// TIA Portal V18 export
// export: Created 2026-06-07T17:38:19.8064699Z, ExportSetting WithDefaults, DisplayName Totally Integrated Automation Portal, DisplayVersion V18, DisplayName TIA Portal Openness, DisplayVersion V18, DisplayName TIA Portal Version Control Interface, DisplayVersion V18, DisplayName STEP 7 Professional, DisplayVersion V18, DisplayName STEP 7 Safety, DisplayVersion V18, DisplayName WinCC Professional, DisplayVersion V18
FUNCTION "FC_PLC2_Mixing" : Void   // FC20, LAD
{ S7_Optimized_Access := 'TRUE' }
VERSION : 0.1
// stored: AutoNumber true, IsIECCheckEnabled false, SetENOAutomatically false, UDAEnableTagReadback false
BEGIN

REGION Network 1: Khóa nút nhấn Start HMI qua Run Enable PLC2
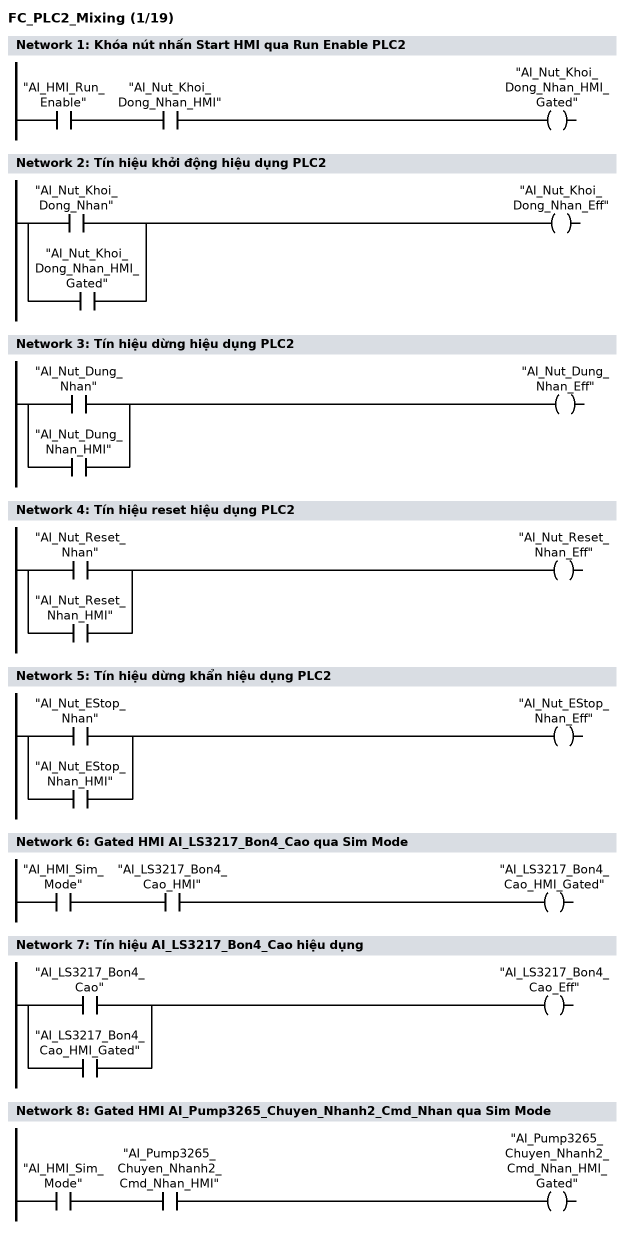
   RUNG wire#powerrail
      Contact( "AI_HMI_Run_Enable" )
      Contact( "AI_Nut_Khoi_Dong_Nhan_HMI" )
      Coil( "AI_Nut_Khoi_Dong_Nhan_HMI_Gated" )
   END_RUNG
   // the same network as SCL:
   "AI_Nut_Khoi_Dong_Nhan_HMI_Gated" := "AI_HMI_Run_Enable" AND "AI_Nut_Khoi_Dong_Nhan_HMI";
END_REGION

REGION Network 2: Tín hiệu khởi động hiệu dụng PLC2
   RUNG wire#powerrail
      Contact( "AI_Nut_Khoi_Dong_Nhan" )
      wire#w1
      Coil( "AI_Nut_Khoi_Dong_Nhan_Eff" )
   END_RUNG
   RUNG wire#powerrail
      Contact( "AI_Nut_Khoi_Dong_Nhan_HMI_Gated" )
   END_RUNG wire#w1
   // the same network as SCL:
   "AI_Nut_Khoi_Dong_Nhan_Eff" := "AI_Nut_Khoi_Dong_Nhan" OR "AI_Nut_Khoi_Dong_Nhan_HMI_Gated";
END_REGION

REGION Network 3: Tín hiệu dừng hiệu dụng PLC2
   RUNG wire#powerrail
      Contact( "AI_Nut_Dung_Nhan" )
      wire#w1
      Coil( "AI_Nut_Dung_Nhan_Eff" )
   END_RUNG
   RUNG wire#powerrail
      Contact( "AI_Nut_Dung_Nhan_HMI" )
   END_RUNG wire#w1
   // the same network as SCL:
   "AI_Nut_Dung_Nhan_Eff" := "AI_Nut_Dung_Nhan" OR "AI_Nut_Dung_Nhan_HMI";
END_REGION

REGION Network 4: Tín hiệu reset hiệu dụng PLC2
   RUNG wire#powerrail
      Contact( "AI_Nut_Reset_Nhan" )
      wire#w1
      Coil( "AI_Nut_Reset_Nhan_Eff" )
   END_RUNG
   RUNG wire#powerrail
      Contact( "AI_Nut_Reset_Nhan_HMI" )
   END_RUNG wire#w1
   // the same network as SCL:
   "AI_Nut_Reset_Nhan_Eff" := "AI_Nut_Reset_Nhan" OR "AI_Nut_Reset_Nhan_HMI";
END_REGION

REGION Network 5: Tín hiệu dừng khẩn hiệu dụng PLC2
   RUNG wire#powerrail
      Contact( "AI_Nut_EStop_Nhan" )
      wire#w1
      Coil( "AI_Nut_EStop_Nhan_Eff" )
   END_RUNG
   RUNG wire#powerrail
      Contact( "AI_Nut_EStop_Nhan_HMI" )
   END_RUNG wire#w1
   // the same network as SCL:
   "AI_Nut_EStop_Nhan_Eff" := "AI_Nut_EStop_Nhan" OR "AI_Nut_EStop_Nhan_HMI";
END_REGION

REGION Network 6: Gated HMI AI_LS3217_Bon4_Cao qua Sim Mode
   RUNG wire#powerrail
      Contact( "AI_HMI_Sim_Mode" )
      Contact( "AI_LS3217_Bon4_Cao_HMI" )
      Coil( "AI_LS3217_Bon4_Cao_HMI_Gated" )
   END_RUNG
   // the same network as SCL:
   "AI_LS3217_Bon4_Cao_HMI_Gated" := "AI_HMI_Sim_Mode" AND "AI_LS3217_Bon4_Cao_HMI";
END_REGION

REGION Network 7: Tín hiệu AI_LS3217_Bon4_Cao hiệu dụng
   RUNG wire#powerrail
      Contact( "AI_LS3217_Bon4_Cao" )
      wire#w1
      Coil( "AI_LS3217_Bon4_Cao_Eff" )
   END_RUNG
   RUNG wire#powerrail
      Contact( "AI_LS3217_Bon4_Cao_HMI_Gated" )
   END_RUNG wire#w1
   // the same network as SCL:
   "AI_LS3217_Bon4_Cao_Eff" := "AI_LS3217_Bon4_Cao" OR "AI_LS3217_Bon4_Cao_HMI_Gated";
END_REGION

REGION Network 8: Gated HMI AI_Pump3265_Chuyen_Nhanh2_Cmd_Nhan qua Sim Mode
   RUNG wire#powerrail
      Contact( "AI_HMI_Sim_Mode" )
      Contact( "AI_Pump3265_Chuyen_Nhanh2_Cmd_Nhan_HMI" )
      Coil( "AI_Pump3265_Chuyen_Nhanh2_Cmd_Nhan_HMI_Gated" )
   END_RUNG
   // the same network as SCL:
   "AI_Pump3265_Chuyen_Nhanh2_Cmd_Nhan_HMI_Gated" := "AI_HMI_Sim_Mode" AND "AI_Pump3265_Chuyen_Nhanh2_Cmd_Nhan_HMI";
END_REGION

REGION Network 9: Tín hiệu AI_Pump3265_Chuyen_Nhanh2_Cmd_Nhan hiệu dụng
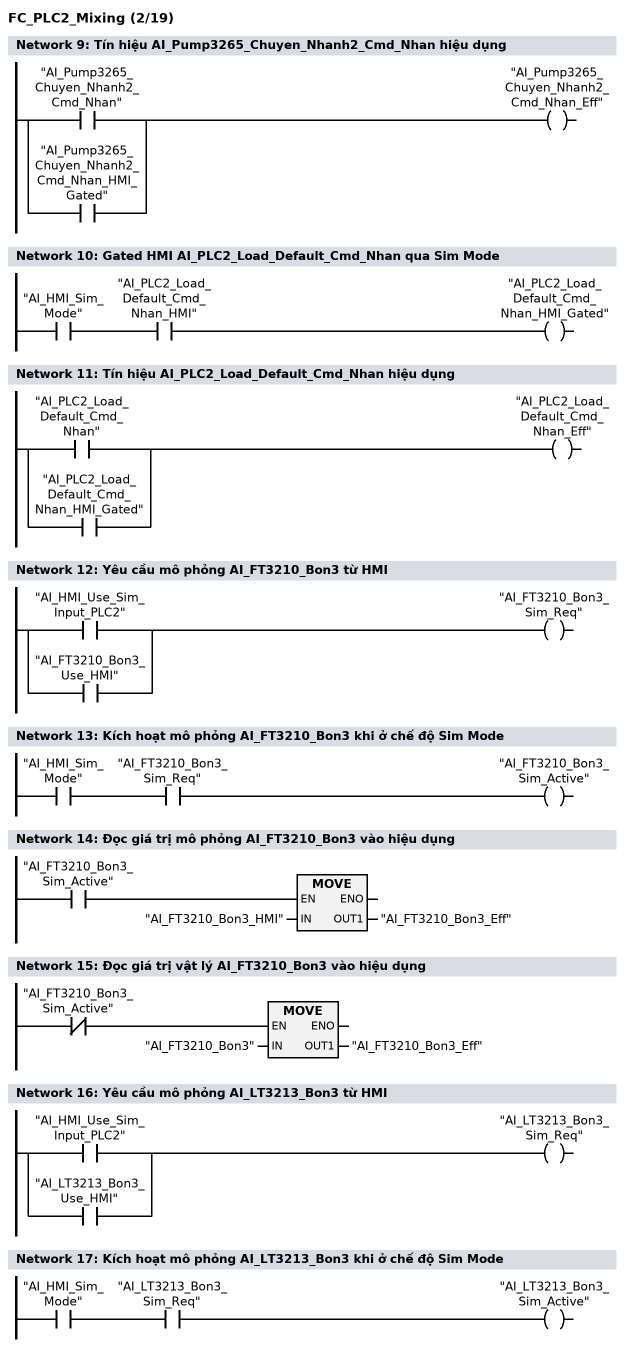
   RUNG wire#powerrail
      Contact( "AI_Pump3265_Chuyen_Nhanh2_Cmd_Nhan" )
      wire#w1
      Coil( "AI_Pump3265_Chuyen_Nhanh2_Cmd_Nhan_Eff" )
   END_RUNG
   RUNG wire#powerrail
      Contact( "AI_Pump3265_Chuyen_Nhanh2_Cmd_Nhan_HMI_Gated" )
   END_RUNG wire#w1
   // the same network as SCL:
   "AI_Pump3265_Chuyen_Nhanh2_Cmd_Nhan_Eff" := "AI_Pump3265_Chuyen_Nhanh2_Cmd_Nhan" OR "AI_Pump3265_Chuyen_Nhanh2_Cmd_Nhan_HMI_Gated";
END_REGION

REGION Network 10: Gated HMI AI_PLC2_Load_Default_Cmd_Nhan qua Sim Mode
   RUNG wire#powerrail
      Contact( "AI_HMI_Sim_Mode" )
      Contact( "AI_PLC2_Load_Default_Cmd_Nhan_HMI" )
      Coil( "AI_PLC2_Load_Default_Cmd_Nhan_HMI_Gated" )
   END_RUNG
   // the same network as SCL:
   "AI_PLC2_Load_Default_Cmd_Nhan_HMI_Gated" := "AI_HMI_Sim_Mode" AND "AI_PLC2_Load_Default_Cmd_Nhan_HMI";
END_REGION

REGION Network 11: Tín hiệu AI_PLC2_Load_Default_Cmd_Nhan hiệu dụng
   RUNG wire#powerrail
      Contact( "AI_PLC2_Load_Default_Cmd_Nhan" )
      wire#w1
      Coil( "AI_PLC2_Load_Default_Cmd_Nhan_Eff" )
   END_RUNG
   RUNG wire#powerrail
      Contact( "AI_PLC2_Load_Default_Cmd_Nhan_HMI_Gated" )
   END_RUNG wire#w1
   // the same network as SCL:
   "AI_PLC2_Load_Default_Cmd_Nhan_Eff" := "AI_PLC2_Load_Default_Cmd_Nhan" OR "AI_PLC2_Load_Default_Cmd_Nhan_HMI_Gated";
END_REGION

REGION Network 12: Yêu cầu mô phỏng AI_FT3210_Bon3 từ HMI
   RUNG wire#powerrail
      Contact( "AI_HMI_Use_Sim_Input_PLC2" )
      wire#w1
      Coil( "AI_FT3210_Bon3_Sim_Req" )
   END_RUNG
   RUNG wire#powerrail
      Contact( "AI_FT3210_Bon3_Use_HMI" )
   END_RUNG wire#w1
   // the same network as SCL:
   "AI_FT3210_Bon3_Sim_Req" := "AI_HMI_Use_Sim_Input_PLC2" OR "AI_FT3210_Bon3_Use_HMI";
END_REGION

REGION Network 13: Kích hoạt mô phỏng AI_FT3210_Bon3 khi ở chế độ Sim Mode
   RUNG wire#powerrail
      Contact( "AI_HMI_Sim_Mode" )
      Contact( "AI_FT3210_Bon3_Sim_Req" )
      Coil( "AI_FT3210_Bon3_Sim_Active" )
   END_RUNG
   // the same network as SCL:
   "AI_FT3210_Bon3_Sim_Active" := "AI_HMI_Sim_Mode" AND "AI_FT3210_Bon3_Sim_Req";
END_REGION

REGION Network 14: Đọc giá trị mô phỏng AI_FT3210_Bon3 vào hiệu dụng
   RUNG wire#powerrail
      Contact( "AI_FT3210_Bon3_Sim_Active" )
      { S7_GenerateENO := "TRUE" } Move(in := "AI_FT3210_Bon3_HMI", out1 => "AI_FT3210_Bon3_Eff")
   END_RUNG
   // the same network as SCL:
   IF "AI_FT3210_Bon3_Sim_Active" THEN "AI_FT3210_Bon3_Eff" := "AI_FT3210_Bon3_HMI"; END_IF;
END_REGION

REGION Network 15: Đọc giá trị vật lý AI_FT3210_Bon3 vào hiệu dụng
   RUNG wire#powerrail
      I_Contact( "AI_FT3210_Bon3_Sim_Active" )
      { S7_GenerateENO := "TRUE" } Move(in := "AI_FT3210_Bon3", out1 => "AI_FT3210_Bon3_Eff")
   END_RUNG
   // the same network as SCL:
   IF NOT "AI_FT3210_Bon3_Sim_Active" THEN "AI_FT3210_Bon3_Eff" := "AI_FT3210_Bon3"; END_IF;
END_REGION

REGION Network 16: Yêu cầu mô phỏng AI_LT3213_Bon3 từ HMI
   RUNG wire#powerrail
      Contact( "AI_HMI_Use_Sim_Input_PLC2" )
      wire#w1
      Coil( "AI_LT3213_Bon3_Sim_Req" )
   END_RUNG
   RUNG wire#powerrail
      Contact( "AI_LT3213_Bon3_Use_HMI" )
   END_RUNG wire#w1
   // the same network as SCL:
   "AI_LT3213_Bon3_Sim_Req" := "AI_HMI_Use_Sim_Input_PLC2" OR "AI_LT3213_Bon3_Use_HMI";
END_REGION

REGION Network 17: Kích hoạt mô phỏng AI_LT3213_Bon3 khi ở chế độ Sim Mode
   RUNG wire#powerrail
      Contact( "AI_HMI_Sim_Mode" )
      Contact( "AI_LT3213_Bon3_Sim_Req" )
      Coil( "AI_LT3213_Bon3_Sim_Active" )
   END_RUNG
   // the same network as SCL:
   "AI_LT3213_Bon3_Sim_Active" := "AI_HMI_Sim_Mode" AND "AI_LT3213_Bon3_Sim_Req";
END_REGION

REGION Network 18: Đọc giá trị mô phỏng AI_LT3213_Bon3 vào hiệu dụng
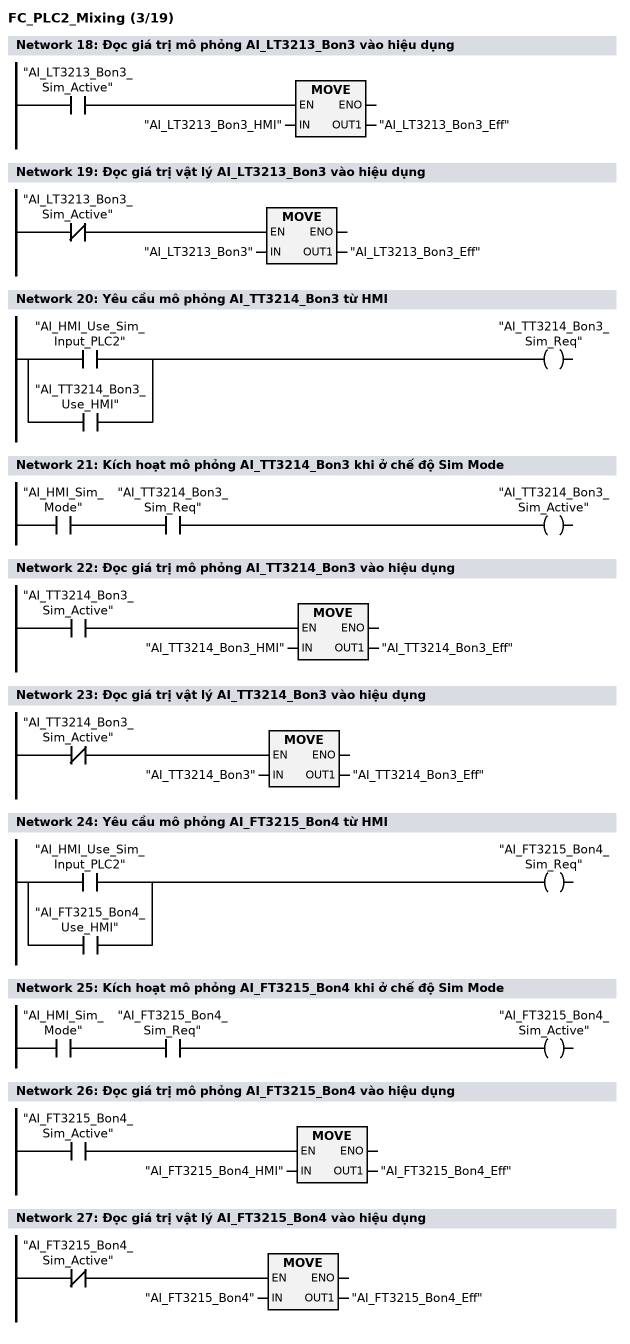
   RUNG wire#powerrail
      Contact( "AI_LT3213_Bon3_Sim_Active" )
      { S7_GenerateENO := "TRUE" } Move(in := "AI_LT3213_Bon3_HMI", out1 => "AI_LT3213_Bon3_Eff")
   END_RUNG
   // the same network as SCL:
   IF "AI_LT3213_Bon3_Sim_Active" THEN "AI_LT3213_Bon3_Eff" := "AI_LT3213_Bon3_HMI"; END_IF;
END_REGION

REGION Network 19: Đọc giá trị vật lý AI_LT3213_Bon3 vào hiệu dụng
   RUNG wire#powerrail
      I_Contact( "AI_LT3213_Bon3_Sim_Active" )
      { S7_GenerateENO := "TRUE" } Move(in := "AI_LT3213_Bon3", out1 => "AI_LT3213_Bon3_Eff")
   END_RUNG
   // the same network as SCL:
   IF NOT "AI_LT3213_Bon3_Sim_Active" THEN "AI_LT3213_Bon3_Eff" := "AI_LT3213_Bon3"; END_IF;
END_REGION

REGION Network 20: Yêu cầu mô phỏng AI_TT3214_Bon3 từ HMI
   RUNG wire#powerrail
      Contact( "AI_HMI_Use_Sim_Input_PLC2" )
      wire#w1
      Coil( "AI_TT3214_Bon3_Sim_Req" )
   END_RUNG
   RUNG wire#powerrail
      Contact( "AI_TT3214_Bon3_Use_HMI" )
   END_RUNG wire#w1
   // the same network as SCL:
   "AI_TT3214_Bon3_Sim_Req" := "AI_HMI_Use_Sim_Input_PLC2" OR "AI_TT3214_Bon3_Use_HMI";
END_REGION

REGION Network 21: Kích hoạt mô phỏng AI_TT3214_Bon3 khi ở chế độ Sim Mode
   RUNG wire#powerrail
      Contact( "AI_HMI_Sim_Mode" )
      Contact( "AI_TT3214_Bon3_Sim_Req" )
      Coil( "AI_TT3214_Bon3_Sim_Active" )
   END_RUNG
   // the same network as SCL:
   "AI_TT3214_Bon3_Sim_Active" := "AI_HMI_Sim_Mode" AND "AI_TT3214_Bon3_Sim_Req";
END_REGION

REGION Network 22: Đọc giá trị mô phỏng AI_TT3214_Bon3 vào hiệu dụng
   RUNG wire#powerrail
      Contact( "AI_TT3214_Bon3_Sim_Active" )
      { S7_GenerateENO := "TRUE" } Move(in := "AI_TT3214_Bon3_HMI", out1 => "AI_TT3214_Bon3_Eff")
   END_RUNG
   // the same network as SCL:
   IF "AI_TT3214_Bon3_Sim_Active" THEN "AI_TT3214_Bon3_Eff" := "AI_TT3214_Bon3_HMI"; END_IF;
END_REGION

REGION Network 23: Đọc giá trị vật lý AI_TT3214_Bon3 vào hiệu dụng
   RUNG wire#powerrail
      I_Contact( "AI_TT3214_Bon3_Sim_Active" )
      { S7_GenerateENO := "TRUE" } Move(in := "AI_TT3214_Bon3", out1 => "AI_TT3214_Bon3_Eff")
   END_RUNG
   // the same network as SCL:
   IF NOT "AI_TT3214_Bon3_Sim_Active" THEN "AI_TT3214_Bon3_Eff" := "AI_TT3214_Bon3"; END_IF;
END_REGION

REGION Network 24: Yêu cầu mô phỏng AI_FT3215_Bon4 từ HMI
   RUNG wire#powerrail
      Contact( "AI_HMI_Use_Sim_Input_PLC2" )
      wire#w1
      Coil( "AI_FT3215_Bon4_Sim_Req" )
   END_RUNG
   RUNG wire#powerrail
      Contact( "AI_FT3215_Bon4_Use_HMI" )
   END_RUNG wire#w1
   // the same network as SCL:
   "AI_FT3215_Bon4_Sim_Req" := "AI_HMI_Use_Sim_Input_PLC2" OR "AI_FT3215_Bon4_Use_HMI";
END_REGION

REGION Network 25: Kích hoạt mô phỏng AI_FT3215_Bon4 khi ở chế độ Sim Mode
   RUNG wire#powerrail
      Contact( "AI_HMI_Sim_Mode" )
      Contact( "AI_FT3215_Bon4_Sim_Req" )
      Coil( "AI_FT3215_Bon4_Sim_Active" )
   END_RUNG
   // the same network as SCL:
   "AI_FT3215_Bon4_Sim_Active" := "AI_HMI_Sim_Mode" AND "AI_FT3215_Bon4_Sim_Req";
END_REGION

REGION Network 26: Đọc giá trị mô phỏng AI_FT3215_Bon4 vào hiệu dụng
   RUNG wire#powerrail
      Contact( "AI_FT3215_Bon4_Sim_Active" )
      { S7_GenerateENO := "TRUE" } Move(in := "AI_FT3215_Bon4_HMI", out1 => "AI_FT3215_Bon4_Eff")
   END_RUNG
   // the same network as SCL:
   IF "AI_FT3215_Bon4_Sim_Active" THEN "AI_FT3215_Bon4_Eff" := "AI_FT3215_Bon4_HMI"; END_IF;
END_REGION

REGION Network 27: Đọc giá trị vật lý AI_FT3215_Bon4 vào hiệu dụng
   RUNG wire#powerrail
      I_Contact( "AI_FT3215_Bon4_Sim_Active" )
      { S7_GenerateENO := "TRUE" } Move(in := "AI_FT3215_Bon4", out1 => "AI_FT3215_Bon4_Eff")
   END_RUNG
   // the same network as SCL:
   IF NOT "AI_FT3215_Bon4_Sim_Active" THEN "AI_FT3215_Bon4_Eff" := "AI_FT3215_Bon4"; END_IF;
END_REGION

REGION Network 28: Yêu cầu mô phỏng AI_FQ3215_Bon4 từ HMI
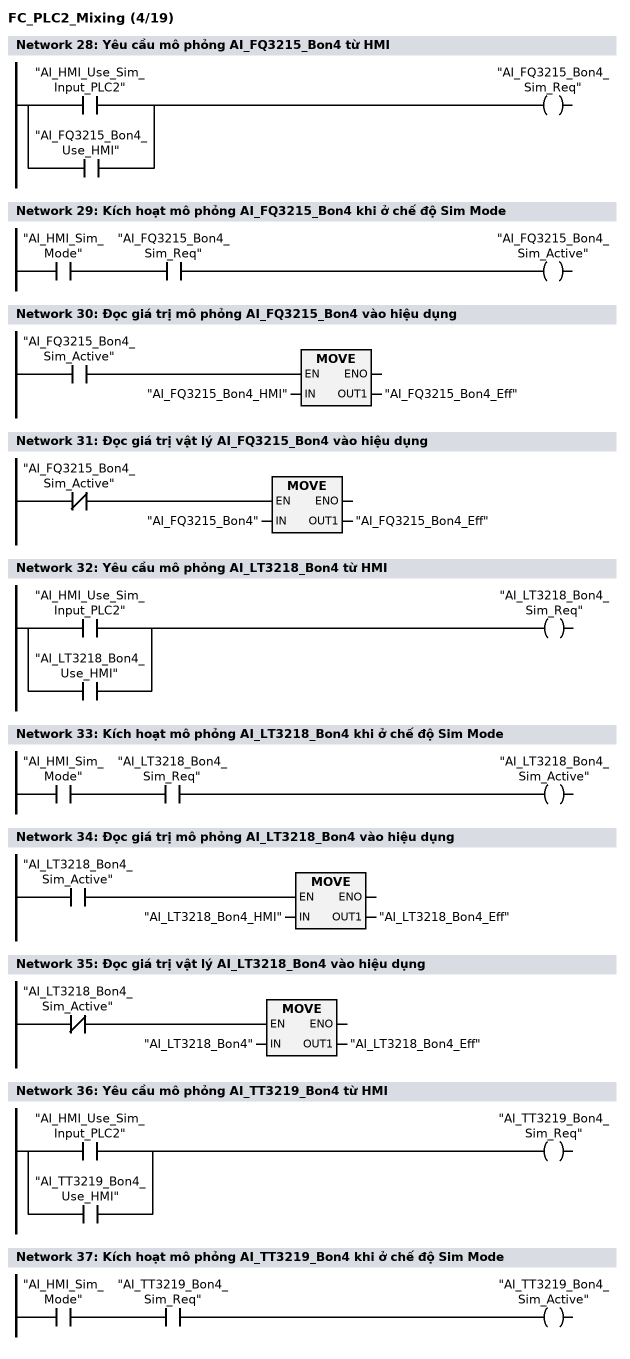
   RUNG wire#powerrail
      Contact( "AI_HMI_Use_Sim_Input_PLC2" )
      wire#w1
      Coil( "AI_FQ3215_Bon4_Sim_Req" )
   END_RUNG
   RUNG wire#powerrail
      Contact( "AI_FQ3215_Bon4_Use_HMI" )
   END_RUNG wire#w1
   // the same network as SCL:
   "AI_FQ3215_Bon4_Sim_Req" := "AI_HMI_Use_Sim_Input_PLC2" OR "AI_FQ3215_Bon4_Use_HMI";
END_REGION

REGION Network 29: Kích hoạt mô phỏng AI_FQ3215_Bon4 khi ở chế độ Sim Mode
   RUNG wire#powerrail
      Contact( "AI_HMI_Sim_Mode" )
      Contact( "AI_FQ3215_Bon4_Sim_Req" )
      Coil( "AI_FQ3215_Bon4_Sim_Active" )
   END_RUNG
   // the same network as SCL:
   "AI_FQ3215_Bon4_Sim_Active" := "AI_HMI_Sim_Mode" AND "AI_FQ3215_Bon4_Sim_Req";
END_REGION

REGION Network 30: Đọc giá trị mô phỏng AI_FQ3215_Bon4 vào hiệu dụng
   RUNG wire#powerrail
      Contact( "AI_FQ3215_Bon4_Sim_Active" )
      { S7_GenerateENO := "TRUE" } Move(in := "AI_FQ3215_Bon4_HMI", out1 => "AI_FQ3215_Bon4_Eff")
   END_RUNG
   // the same network as SCL:
   IF "AI_FQ3215_Bon4_Sim_Active" THEN "AI_FQ3215_Bon4_Eff" := "AI_FQ3215_Bon4_HMI"; END_IF;
END_REGION

REGION Network 31: Đọc giá trị vật lý AI_FQ3215_Bon4 vào hiệu dụng
   RUNG wire#powerrail
      I_Contact( "AI_FQ3215_Bon4_Sim_Active" )
      { S7_GenerateENO := "TRUE" } Move(in := "AI_FQ3215_Bon4", out1 => "AI_FQ3215_Bon4_Eff")
   END_RUNG
   // the same network as SCL:
   IF NOT "AI_FQ3215_Bon4_Sim_Active" THEN "AI_FQ3215_Bon4_Eff" := "AI_FQ3215_Bon4"; END_IF;
END_REGION

REGION Network 32: Yêu cầu mô phỏng AI_LT3218_Bon4 từ HMI
   RUNG wire#powerrail
      Contact( "AI_HMI_Use_Sim_Input_PLC2" )
      wire#w1
      Coil( "AI_LT3218_Bon4_Sim_Req" )
   END_RUNG
   RUNG wire#powerrail
      Contact( "AI_LT3218_Bon4_Use_HMI" )
   END_RUNG wire#w1
   // the same network as SCL:
   "AI_LT3218_Bon4_Sim_Req" := "AI_HMI_Use_Sim_Input_PLC2" OR "AI_LT3218_Bon4_Use_HMI";
END_REGION

REGION Network 33: Kích hoạt mô phỏng AI_LT3218_Bon4 khi ở chế độ Sim Mode
   RUNG wire#powerrail
      Contact( "AI_HMI_Sim_Mode" )
      Contact( "AI_LT3218_Bon4_Sim_Req" )
      Coil( "AI_LT3218_Bon4_Sim_Active" )
   END_RUNG
   // the same network as SCL:
   "AI_LT3218_Bon4_Sim_Active" := "AI_HMI_Sim_Mode" AND "AI_LT3218_Bon4_Sim_Req";
END_REGION

REGION Network 34: Đọc giá trị mô phỏng AI_LT3218_Bon4 vào hiệu dụng
   RUNG wire#powerrail
      Contact( "AI_LT3218_Bon4_Sim_Active" )
      { S7_GenerateENO := "TRUE" } Move(in := "AI_LT3218_Bon4_HMI", out1 => "AI_LT3218_Bon4_Eff")
   END_RUNG
   // the same network as SCL:
   IF "AI_LT3218_Bon4_Sim_Active" THEN "AI_LT3218_Bon4_Eff" := "AI_LT3218_Bon4_HMI"; END_IF;
END_REGION

REGION Network 35: Đọc giá trị vật lý AI_LT3218_Bon4 vào hiệu dụng
   RUNG wire#powerrail
      I_Contact( "AI_LT3218_Bon4_Sim_Active" )
      { S7_GenerateENO := "TRUE" } Move(in := "AI_LT3218_Bon4", out1 => "AI_LT3218_Bon4_Eff")
   END_RUNG
   // the same network as SCL:
   IF NOT "AI_LT3218_Bon4_Sim_Active" THEN "AI_LT3218_Bon4_Eff" := "AI_LT3218_Bon4"; END_IF;
END_REGION

REGION Network 36: Yêu cầu mô phỏng AI_TT3219_Bon4 từ HMI
   RUNG wire#powerrail
      Contact( "AI_HMI_Use_Sim_Input_PLC2" )
      wire#w1
      Coil( "AI_TT3219_Bon4_Sim_Req" )
   END_RUNG
   RUNG wire#powerrail
      Contact( "AI_TT3219_Bon4_Use_HMI" )
   END_RUNG wire#w1
   // the same network as SCL:
   "AI_TT3219_Bon4_Sim_Req" := "AI_HMI_Use_Sim_Input_PLC2" OR "AI_TT3219_Bon4_Use_HMI";
END_REGION

REGION Network 37: Kích hoạt mô phỏng AI_TT3219_Bon4 khi ở chế độ Sim Mode
   RUNG wire#powerrail
      Contact( "AI_HMI_Sim_Mode" )
      Contact( "AI_TT3219_Bon4_Sim_Req" )
      Coil( "AI_TT3219_Bon4_Sim_Active" )
   END_RUNG
   // the same network as SCL:
   "AI_TT3219_Bon4_Sim_Active" := "AI_HMI_Sim_Mode" AND "AI_TT3219_Bon4_Sim_Req";
END_REGION

REGION Network 38: Đọc giá trị mô phỏng AI_TT3219_Bon4 vào hiệu dụng
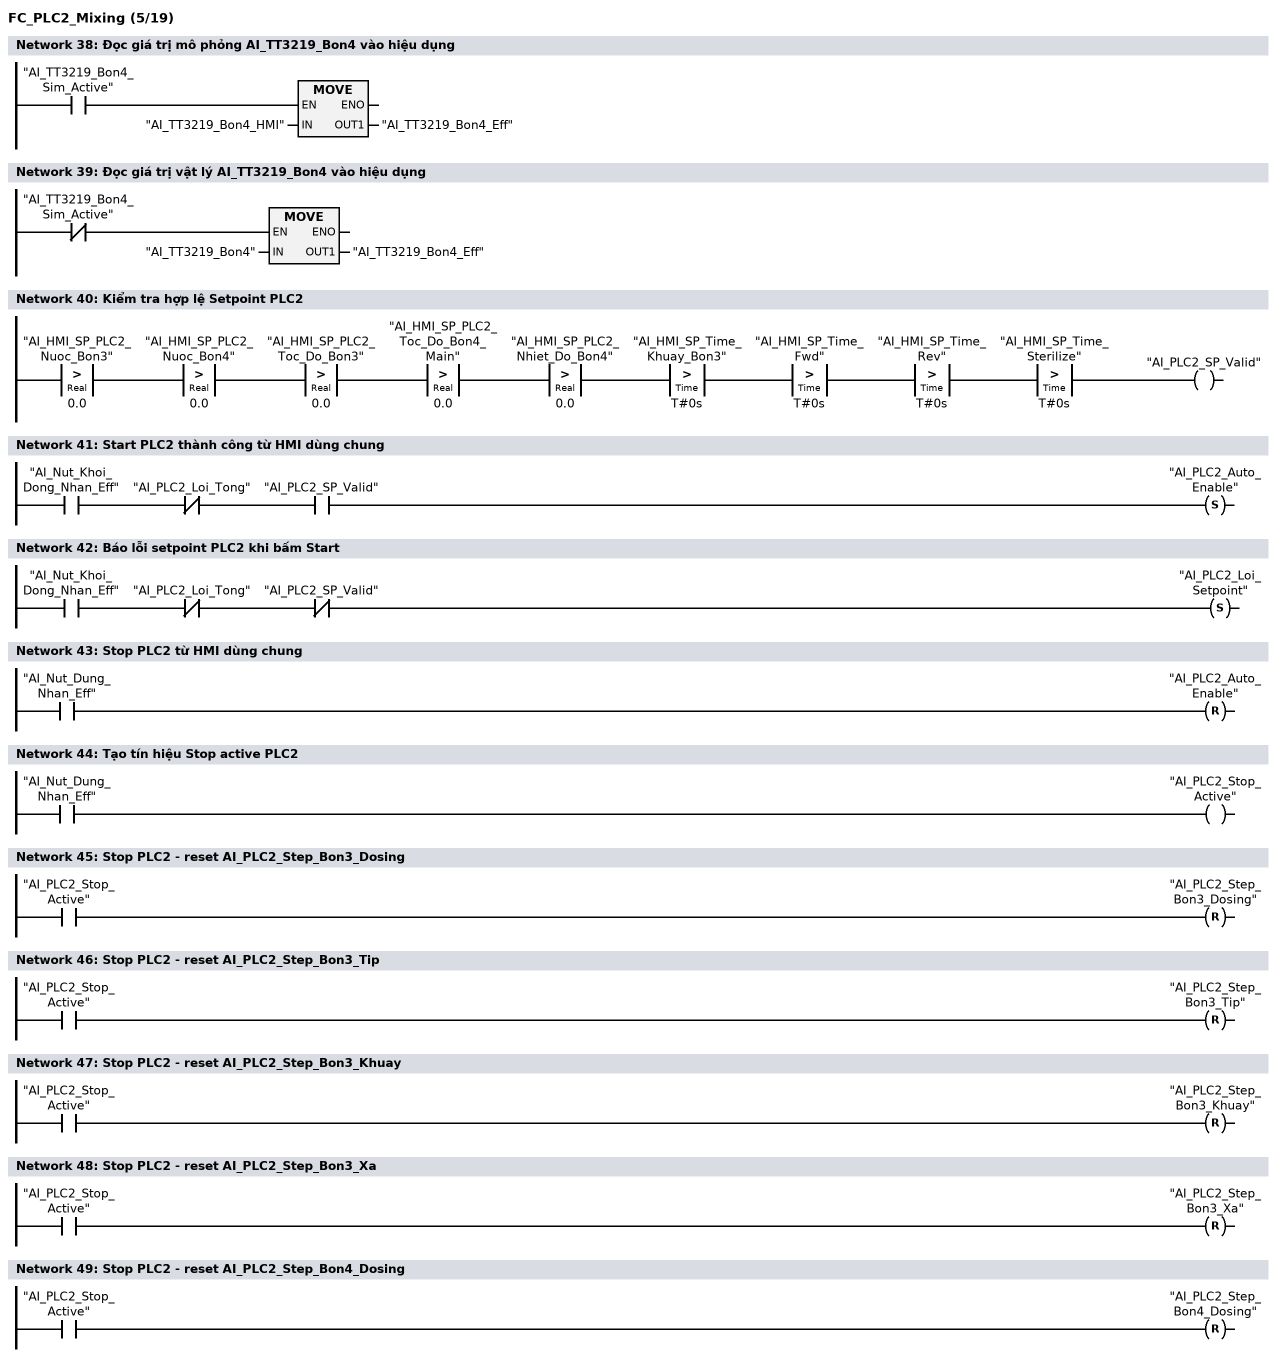
   RUNG wire#powerrail
      Contact( "AI_TT3219_Bon4_Sim_Active" )
      { S7_GenerateENO := "TRUE" } Move(in := "AI_TT3219_Bon4_HMI", out1 => "AI_TT3219_Bon4_Eff")
   END_RUNG
   // the same network as SCL:
   IF "AI_TT3219_Bon4_Sim_Active" THEN "AI_TT3219_Bon4_Eff" := "AI_TT3219_Bon4_HMI"; END_IF;
END_REGION

REGION Network 39: Đọc giá trị vật lý AI_TT3219_Bon4 vào hiệu dụng
   RUNG wire#powerrail
      I_Contact( "AI_TT3219_Bon4_Sim_Active" )
      { S7_GenerateENO := "TRUE" } Move(in := "AI_TT3219_Bon4", out1 => "AI_TT3219_Bon4_Eff")
   END_RUNG
   // the same network as SCL:
   IF NOT "AI_TT3219_Bon4_Sim_Active" THEN "AI_TT3219_Bon4_Eff" := "AI_TT3219_Bon4"; END_IF;
END_REGION

REGION Network 40: Kiểm tra hợp lệ Setpoint PLC2
   RUNG wire#powerrail
      { S7_Templates := "SrcType := Real" } GT_Contact(in1 := "AI_HMI_SP_PLC2_Nuoc_Bon3", in2 := 0.0)
      { S7_Templates := "SrcType := Real" } GT_Contact(in1 := "AI_HMI_SP_PLC2_Nuoc_Bon4", in2 := 0.0)
      { S7_Templates := "SrcType := Real" } GT_Contact(in1 := "AI_HMI_SP_PLC2_Toc_Do_Bon3", in2 := 0.0)
      { S7_Templates := "SrcType := Real" } GT_Contact(in1 := "AI_HMI_SP_PLC2_Toc_Do_Bon4_Main", in2 := 0.0)
      { S7_Templates := "SrcType := Real" } GT_Contact(in1 := "AI_HMI_SP_PLC2_Nhiet_Do_Bon4", in2 := 0.0)
      { S7_Templates := "SrcType := Time" } GT_Contact(in1 := "AI_HMI_SP_Time_Khuay_Bon3", in2 := T#0s)
      { S7_Templates := "SrcType := Time" } GT_Contact(in1 := "AI_HMI_SP_Time_Fwd", in2 := T#0s)
      { S7_Templates := "SrcType := Time" } GT_Contact(in1 := "AI_HMI_SP_Time_Rev", in2 := T#0s)
      { S7_Templates := "SrcType := Time" } GT_Contact(in1 := "AI_HMI_SP_Time_Sterilize", in2 := T#0s)
      Coil( "AI_PLC2_SP_Valid" )
   END_RUNG
   // the same network as SCL:
   "AI_PLC2_SP_Valid" := ("AI_HMI_SP_PLC2_Nuoc_Bon3" > 0.0) AND ("AI_HMI_SP_PLC2_Nuoc_Bon4" > 0.0) AND ("AI_HMI_SP_PLC2_Toc_Do_Bon3" > 0.0) AND ("AI_HMI_SP_PLC2_Toc_Do_Bon4_Main" > 0.0) AND ("AI_HMI_SP_PLC2_Nhiet_Do_Bon4" > 0.0) AND ("AI_HMI_SP_Time_Khuay_Bon3" > T#0s) AND ("AI_HMI_SP_Time_Fwd" > T#0s) AND ("AI_HMI_SP_Time_Rev" > T#0s) AND ("AI_HMI_SP_Time_Sterilize" > T#0s);
END_REGION

REGION Network 41: Start PLC2 thành công từ HMI dùng chung
   RUNG wire#powerrail
      Contact( "AI_Nut_Khoi_Dong_Nhan_Eff" )
      I_Contact( "AI_PLC2_Loi_Tong" )
      Contact( "AI_PLC2_SP_Valid" )
      S_Coil( "AI_PLC2_Auto_Enable" )
   END_RUNG
   // the same network as SCL:
   IF "AI_Nut_Khoi_Dong_Nhan_Eff" AND NOT "AI_PLC2_Loi_Tong" AND "AI_PLC2_SP_Valid" THEN
       "AI_PLC2_Auto_Enable" := TRUE;
   END_IF;
END_REGION

REGION Network 42: Báo lỗi setpoint PLC2 khi bấm Start
   RUNG wire#powerrail
      Contact( "AI_Nut_Khoi_Dong_Nhan_Eff" )
      I_Contact( "AI_PLC2_Loi_Tong" )
      I_Contact( "AI_PLC2_SP_Valid" )
      S_Coil( "AI_PLC2_Loi_Setpoint" )
   END_RUNG
   // the same network as SCL:
   IF "AI_Nut_Khoi_Dong_Nhan_Eff" AND NOT "AI_PLC2_Loi_Tong" AND NOT "AI_PLC2_SP_Valid" THEN
       "AI_PLC2_Loi_Setpoint" := TRUE;
   END_IF;
END_REGION

REGION Network 43: Stop PLC2 từ HMI dùng chung
   RUNG wire#powerrail
      Contact( "AI_Nut_Dung_Nhan_Eff" )
      R_Coil( "AI_PLC2_Auto_Enable" )
   END_RUNG
   // the same network as SCL:
   IF "AI_Nut_Dung_Nhan_Eff" THEN "AI_PLC2_Auto_Enable" := FALSE; END_IF;
END_REGION

REGION Network 44: Tạo tín hiệu Stop active PLC2
   RUNG wire#powerrail
      Contact( "AI_Nut_Dung_Nhan_Eff" )
      Coil( "AI_PLC2_Stop_Active" )
   END_RUNG
   // the same network as SCL:
   "AI_PLC2_Stop_Active" := "AI_Nut_Dung_Nhan_Eff";
END_REGION

REGION Network 45: Stop PLC2 - reset AI_PLC2_Step_Bon3_Dosing
   RUNG wire#powerrail
      Contact( "AI_PLC2_Stop_Active" )
      R_Coil( "AI_PLC2_Step_Bon3_Dosing" )
   END_RUNG
   // the same network as SCL:
   IF "AI_PLC2_Stop_Active" THEN "AI_PLC2_Step_Bon3_Dosing" := FALSE; END_IF;
END_REGION

REGION Network 46: Stop PLC2 - reset AI_PLC2_Step_Bon3_Tip
   RUNG wire#powerrail
      Contact( "AI_PLC2_Stop_Active" )
      R_Coil( "AI_PLC2_Step_Bon3_Tip" )
   END_RUNG
   // the same network as SCL:
   IF "AI_PLC2_Stop_Active" THEN "AI_PLC2_Step_Bon3_Tip" := FALSE; END_IF;
END_REGION

REGION Network 47: Stop PLC2 - reset AI_PLC2_Step_Bon3_Khuay
   RUNG wire#powerrail
      Contact( "AI_PLC2_Stop_Active" )
      R_Coil( "AI_PLC2_Step_Bon3_Khuay" )
   END_RUNG
   // the same network as SCL:
   IF "AI_PLC2_Stop_Active" THEN "AI_PLC2_Step_Bon3_Khuay" := FALSE; END_IF;
END_REGION

REGION Network 48: Stop PLC2 - reset AI_PLC2_Step_Bon3_Xa
   RUNG wire#powerrail
      Contact( "AI_PLC2_Stop_Active" )
      R_Coil( "AI_PLC2_Step_Bon3_Xa" )
   END_RUNG
   // the same network as SCL:
   IF "AI_PLC2_Stop_Active" THEN "AI_PLC2_Step_Bon3_Xa" := FALSE; END_IF;
END_REGION

REGION Network 49: Stop PLC2 - reset AI_PLC2_Step_Bon4_Dosing
   RUNG wire#powerrail
      Contact( "AI_PLC2_Stop_Active" )
      R_Coil( "AI_PLC2_Step_Bon4_Dosing" )
   END_RUNG
   // the same network as SCL:
   IF "AI_PLC2_Stop_Active" THEN "AI_PLC2_Step_Bon4_Dosing" := FALSE; END_IF;
END_REGION

REGION Network 50: Stop PLC2 - reset AI_PLC2_Step_Bon4_Tip
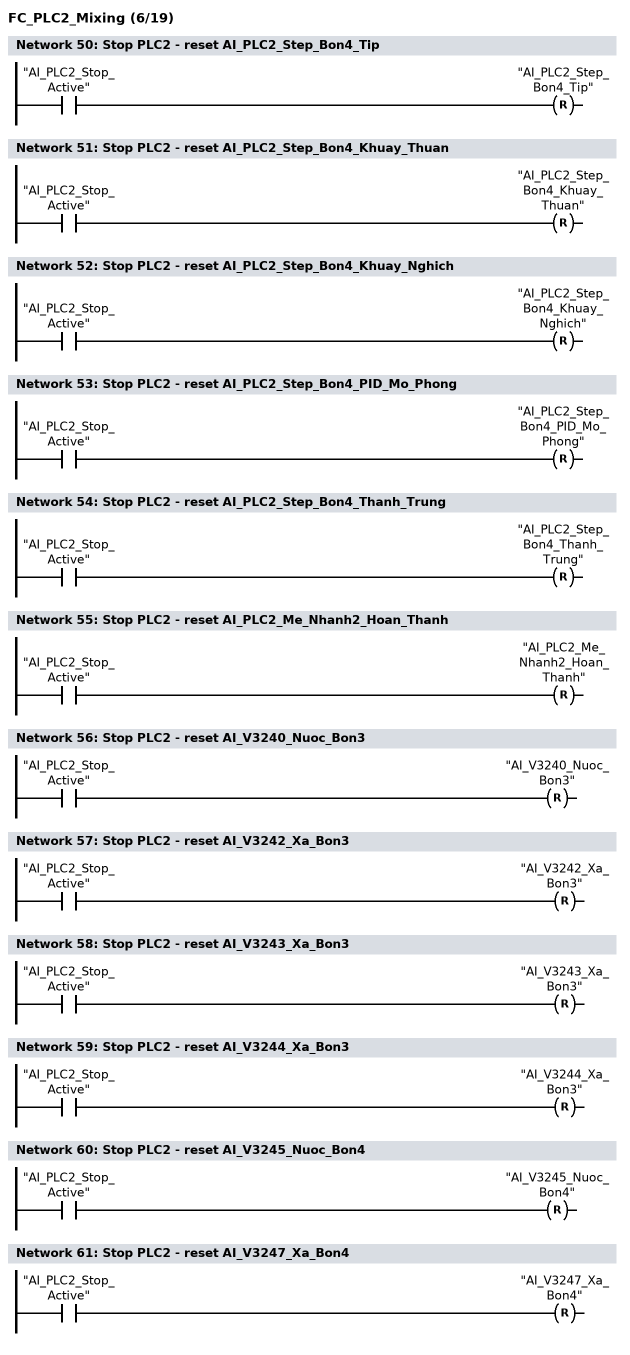
   RUNG wire#powerrail
      Contact( "AI_PLC2_Stop_Active" )
      R_Coil( "AI_PLC2_Step_Bon4_Tip" )
   END_RUNG
   // the same network as SCL:
   IF "AI_PLC2_Stop_Active" THEN "AI_PLC2_Step_Bon4_Tip" := FALSE; END_IF;
END_REGION

REGION Network 51: Stop PLC2 - reset AI_PLC2_Step_Bon4_Khuay_Thuan
   RUNG wire#powerrail
      Contact( "AI_PLC2_Stop_Active" )
      R_Coil( "AI_PLC2_Step_Bon4_Khuay_Thuan" )
   END_RUNG
   // the same network as SCL:
   IF "AI_PLC2_Stop_Active" THEN "AI_PLC2_Step_Bon4_Khuay_Thuan" := FALSE; END_IF;
END_REGION

REGION Network 52: Stop PLC2 - reset AI_PLC2_Step_Bon4_Khuay_Nghich
   RUNG wire#powerrail
      Contact( "AI_PLC2_Stop_Active" )
      R_Coil( "AI_PLC2_Step_Bon4_Khuay_Nghich" )
   END_RUNG
   // the same network as SCL:
   IF "AI_PLC2_Stop_Active" THEN "AI_PLC2_Step_Bon4_Khuay_Nghich" := FALSE; END_IF;
END_REGION

REGION Network 53: Stop PLC2 - reset AI_PLC2_Step_Bon4_PID_Mo_Phong
   RUNG wire#powerrail
      Contact( "AI_PLC2_Stop_Active" )
      R_Coil( "AI_PLC2_Step_Bon4_PID_Mo_Phong" )
   END_RUNG
   // the same network as SCL:
   IF "AI_PLC2_Stop_Active" THEN "AI_PLC2_Step_Bon4_PID_Mo_Phong" := FALSE; END_IF;
END_REGION

REGION Network 54: Stop PLC2 - reset AI_PLC2_Step_Bon4_Thanh_Trung
   RUNG wire#powerrail
      Contact( "AI_PLC2_Stop_Active" )
      R_Coil( "AI_PLC2_Step_Bon4_Thanh_Trung" )
   END_RUNG
   // the same network as SCL:
   IF "AI_PLC2_Stop_Active" THEN "AI_PLC2_Step_Bon4_Thanh_Trung" := FALSE; END_IF;
END_REGION

REGION Network 55: Stop PLC2 - reset AI_PLC2_Me_Nhanh2_Hoan_Thanh
   RUNG wire#powerrail
      Contact( "AI_PLC2_Stop_Active" )
      R_Coil( "AI_PLC2_Me_Nhanh2_Hoan_Thanh" )
   END_RUNG
   // the same network as SCL:
   IF "AI_PLC2_Stop_Active" THEN "AI_PLC2_Me_Nhanh2_Hoan_Thanh" := FALSE; END_IF;
END_REGION

REGION Network 56: Stop PLC2 - reset AI_V3240_Nuoc_Bon3
   RUNG wire#powerrail
      Contact( "AI_PLC2_Stop_Active" )
      R_Coil( "AI_V3240_Nuoc_Bon3" )
   END_RUNG
   // the same network as SCL:
   IF "AI_PLC2_Stop_Active" THEN "AI_V3240_Nuoc_Bon3" := FALSE; END_IF;
END_REGION

REGION Network 57: Stop PLC2 - reset AI_V3242_Xa_Bon3
   RUNG wire#powerrail
      Contact( "AI_PLC2_Stop_Active" )
      R_Coil( "AI_V3242_Xa_Bon3" )
   END_RUNG
   // the same network as SCL:
   IF "AI_PLC2_Stop_Active" THEN "AI_V3242_Xa_Bon3" := FALSE; END_IF;
END_REGION

REGION Network 58: Stop PLC2 - reset AI_V3243_Xa_Bon3
   RUNG wire#powerrail
      Contact( "AI_PLC2_Stop_Active" )
      R_Coil( "AI_V3243_Xa_Bon3" )
   END_RUNG
   // the same network as SCL:
   IF "AI_PLC2_Stop_Active" THEN "AI_V3243_Xa_Bon3" := FALSE; END_IF;
END_REGION

REGION Network 59: Stop PLC2 - reset AI_V3244_Xa_Bon3
   RUNG wire#powerrail
      Contact( "AI_PLC2_Stop_Active" )
      R_Coil( "AI_V3244_Xa_Bon3" )
   END_RUNG
   // the same network as SCL:
   IF "AI_PLC2_Stop_Active" THEN "AI_V3244_Xa_Bon3" := FALSE; END_IF;
END_REGION

REGION Network 60: Stop PLC2 - reset AI_V3245_Nuoc_Bon4
   RUNG wire#powerrail
      Contact( "AI_PLC2_Stop_Active" )
      R_Coil( "AI_V3245_Nuoc_Bon4" )
   END_RUNG
   // the same network as SCL:
   IF "AI_PLC2_Stop_Active" THEN "AI_V3245_Nuoc_Bon4" := FALSE; END_IF;
END_REGION

REGION Network 61: Stop PLC2 - reset AI_V3247_Xa_Bon4
   RUNG wire#powerrail
      Contact( "AI_PLC2_Stop_Active" )
      R_Coil( "AI_V3247_Xa_Bon4" )
   END_RUNG
   // the same network as SCL:
   IF "AI_PLC2_Stop_Active" THEN "AI_V3247_Xa_Bon4" := FALSE; END_IF;
END_REGION

REGION Network 62: Stop PLC2 - reset AI_V3248_Xa_Bon4
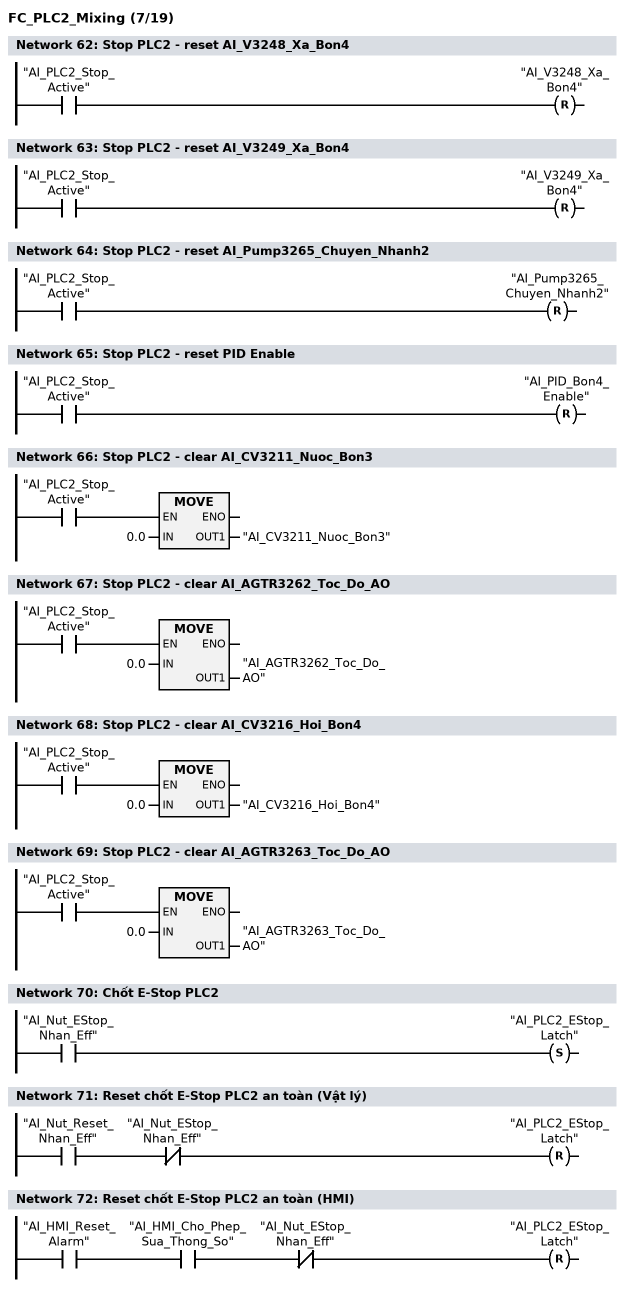
   RUNG wire#powerrail
      Contact( "AI_PLC2_Stop_Active" )
      R_Coil( "AI_V3248_Xa_Bon4" )
   END_RUNG
   // the same network as SCL:
   IF "AI_PLC2_Stop_Active" THEN "AI_V3248_Xa_Bon4" := FALSE; END_IF;
END_REGION

REGION Network 63: Stop PLC2 - reset AI_V3249_Xa_Bon4
   RUNG wire#powerrail
      Contact( "AI_PLC2_Stop_Active" )
      R_Coil( "AI_V3249_Xa_Bon4" )
   END_RUNG
   // the same network as SCL:
   IF "AI_PLC2_Stop_Active" THEN "AI_V3249_Xa_Bon4" := FALSE; END_IF;
END_REGION

REGION Network 64: Stop PLC2 - reset AI_Pump3265_Chuyen_Nhanh2
   RUNG wire#powerrail
      Contact( "AI_PLC2_Stop_Active" )
      R_Coil( "AI_Pump3265_Chuyen_Nhanh2" )
   END_RUNG
   // the same network as SCL:
   IF "AI_PLC2_Stop_Active" THEN "AI_Pump3265_Chuyen_Nhanh2" := FALSE; END_IF;
END_REGION

REGION Network 65: Stop PLC2 - reset PID Enable
   RUNG wire#powerrail
      Contact( "AI_PLC2_Stop_Active" )
      R_Coil( "AI_PID_Bon4_Enable" )
   END_RUNG
   // the same network as SCL:
   IF "AI_PLC2_Stop_Active" THEN "AI_PID_Bon4_Enable" := FALSE; END_IF;
END_REGION

REGION Network 66: Stop PLC2 - clear AI_CV3211_Nuoc_Bon3
   RUNG wire#powerrail
      Contact( "AI_PLC2_Stop_Active" )
      { S7_GenerateENO := "TRUE" } Move(in := 0.0, out1 => "AI_CV3211_Nuoc_Bon3")
   END_RUNG
   // the same network as SCL:
   IF "AI_PLC2_Stop_Active" THEN "AI_CV3211_Nuoc_Bon3" := 0.0; END_IF;
END_REGION

REGION Network 67: Stop PLC2 - clear AI_AGTR3262_Toc_Do_AO
   RUNG wire#powerrail
      Contact( "AI_PLC2_Stop_Active" )
      { S7_GenerateENO := "TRUE" } Move(in := 0.0, out1 => "AI_AGTR3262_Toc_Do_AO")
   END_RUNG
   // the same network as SCL:
   IF "AI_PLC2_Stop_Active" THEN "AI_AGTR3262_Toc_Do_AO" := 0.0; END_IF;
END_REGION

REGION Network 68: Stop PLC2 - clear AI_CV3216_Hoi_Bon4
   RUNG wire#powerrail
      Contact( "AI_PLC2_Stop_Active" )
      { S7_GenerateENO := "TRUE" } Move(in := 0.0, out1 => "AI_CV3216_Hoi_Bon4")
   END_RUNG
   // the same network as SCL:
   IF "AI_PLC2_Stop_Active" THEN "AI_CV3216_Hoi_Bon4" := 0.0; END_IF;
END_REGION

REGION Network 69: Stop PLC2 - clear AI_AGTR3263_Toc_Do_AO
   RUNG wire#powerrail
      Contact( "AI_PLC2_Stop_Active" )
      { S7_GenerateENO := "TRUE" } Move(in := 0.0, out1 => "AI_AGTR3263_Toc_Do_AO")
   END_RUNG
   // the same network as SCL:
   IF "AI_PLC2_Stop_Active" THEN "AI_AGTR3263_Toc_Do_AO" := 0.0; END_IF;
END_REGION

REGION Network 70: Chốt E-Stop PLC2
   RUNG wire#powerrail
      Contact( "AI_Nut_EStop_Nhan_Eff" )
      S_Coil( "AI_PLC2_EStop_Latch" )
   END_RUNG
   // the same network as SCL:
   IF "AI_Nut_EStop_Nhan_Eff" THEN "AI_PLC2_EStop_Latch" := TRUE; END_IF;
END_REGION

REGION Network 71: Reset chốt E-Stop PLC2 an toàn (Vật lý)
   RUNG wire#powerrail
      Contact( "AI_Nut_Reset_Nhan_Eff" )
      I_Contact( "AI_Nut_EStop_Nhan_Eff" )
      R_Coil( "AI_PLC2_EStop_Latch" )
   END_RUNG
   // the same network as SCL:
   IF "AI_Nut_Reset_Nhan_Eff" AND NOT "AI_Nut_EStop_Nhan_Eff" THEN "AI_PLC2_EStop_Latch" := FALSE; END_IF;
END_REGION

REGION Network 72: Reset chốt E-Stop PLC2 an toàn (HMI)
   RUNG wire#powerrail
      Contact( "AI_HMI_Reset_Alarm" )
      Contact( "AI_HMI_Cho_Phep_Sua_Thong_So" )
      I_Contact( "AI_Nut_EStop_Nhan_Eff" )
      R_Coil( "AI_PLC2_EStop_Latch" )
   END_RUNG
   // the same network as SCL:
   IF "AI_HMI_Reset_Alarm" AND "AI_HMI_Cho_Phep_Sua_Thong_So" AND NOT "AI_Nut_EStop_Nhan_Eff" THEN
       "AI_PLC2_EStop_Latch" := FALSE;
   END_IF;
END_REGION

REGION Network 73: Mất truyền thông PLC2
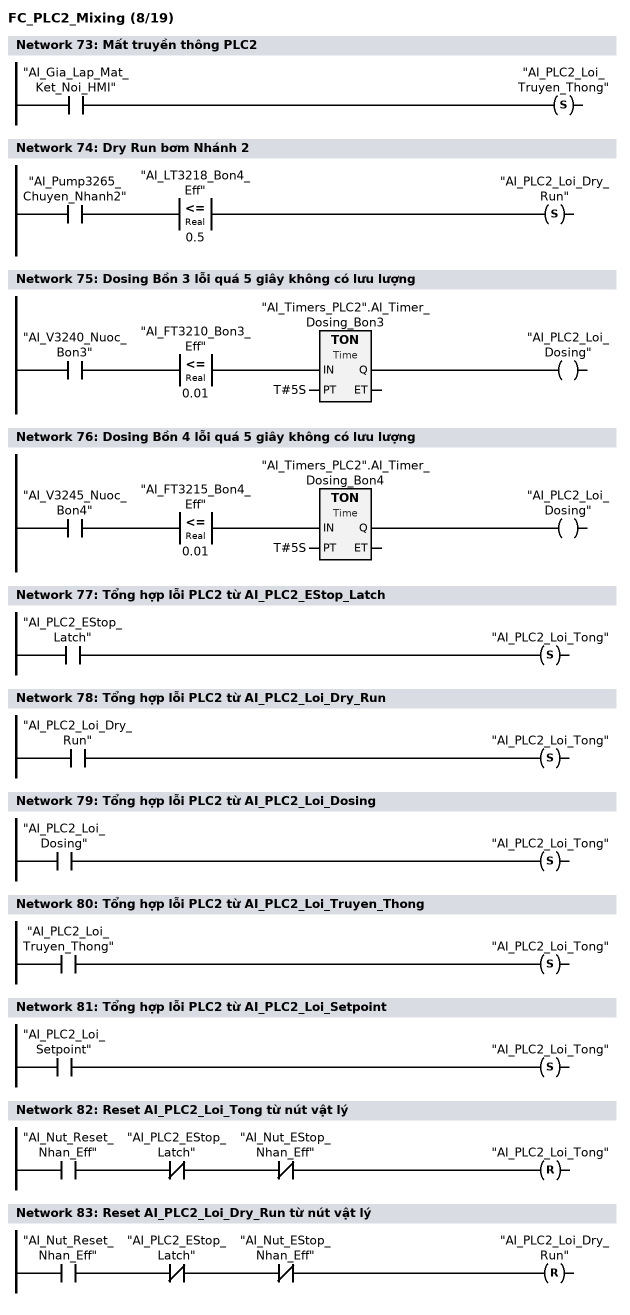
   RUNG wire#powerrail
      Contact( "AI_Gia_Lap_Mat_Ket_Noi_HMI" )
      S_Coil( "AI_PLC2_Loi_Truyen_Thong" )
   END_RUNG
   // the same network as SCL:
   IF "AI_Gia_Lap_Mat_Ket_Noi_HMI" THEN "AI_PLC2_Loi_Truyen_Thong" := TRUE; END_IF;
END_REGION

REGION Network 74: Dry Run bơm Nhánh 2
   RUNG wire#powerrail
      Contact( "AI_Pump3265_Chuyen_Nhanh2" )
      { S7_Templates := "SrcType := Real" } LE_Contact(in1 := "AI_LT3218_Bon4_Eff", in2 := 0.5)
      S_Coil( "AI_PLC2_Loi_Dry_Run" )
   END_RUNG
   // the same network as SCL:
   IF "AI_Pump3265_Chuyen_Nhanh2" AND ("AI_LT3218_Bon4_Eff" <= 0.5) THEN
       "AI_PLC2_Loi_Dry_Run" := TRUE;
   END_IF;
END_REGION

REGION Network 75: Dosing Bồn 3 lỗi quá 5 giây không có lưu lượng
   RUNG wire#powerrail
      Contact( "AI_V3240_Nuoc_Bon3" )
      { S7_Templates := "SrcType := Real" } LE_Contact(in1 := "AI_FT3210_Bon3_Eff", in2 := 0.01)
      { S7_Templates := "time_type := Time" } "AI_Timers_PLC2".AI_Timer_Dosing_Bon3.TON(pt := T#5S, et =>)
      Coil( "AI_PLC2_Loi_Dosing" )
   END_RUNG
   // the same network as SCL:
   "AI_Timers_PLC2".AI_Timer_Dosing_Bon3.TON(IN := "AI_V3240_Nuoc_Bon3" AND ("AI_FT3210_Bon3_Eff" <= 0.01),
                           PT := T#5S);
   "AI_PLC2_Loi_Dosing" := "AI_Timers_PLC2".AI_Timer_Dosing_Bon3.Q;
END_REGION

REGION Network 76: Dosing Bồn 4 lỗi quá 5 giây không có lưu lượng
   RUNG wire#powerrail
      Contact( "AI_V3245_Nuoc_Bon4" )
      { S7_Templates := "SrcType := Real" } LE_Contact(in1 := "AI_FT3215_Bon4_Eff", in2 := 0.01)
      { S7_Templates := "time_type := Time" } "AI_Timers_PLC2".AI_Timer_Dosing_Bon4.TON(pt := T#5S, et =>)
      Coil( "AI_PLC2_Loi_Dosing" )
   END_RUNG
   // the same network as SCL:
   "AI_Timers_PLC2".AI_Timer_Dosing_Bon4.TON(IN := "AI_V3245_Nuoc_Bon4" AND ("AI_FT3215_Bon4_Eff" <= 0.01),
                           PT := T#5S);
   "AI_PLC2_Loi_Dosing" := "AI_Timers_PLC2".AI_Timer_Dosing_Bon4.Q;
END_REGION

REGION Network 77: Tổng hợp lỗi PLC2 từ AI_PLC2_EStop_Latch
   RUNG wire#powerrail
      Contact( "AI_PLC2_EStop_Latch" )
      S_Coil( "AI_PLC2_Loi_Tong" )
   END_RUNG
   // the same network as SCL:
   IF "AI_PLC2_EStop_Latch" THEN "AI_PLC2_Loi_Tong" := TRUE; END_IF;
END_REGION

REGION Network 78: Tổng hợp lỗi PLC2 từ AI_PLC2_Loi_Dry_Run
   RUNG wire#powerrail
      Contact( "AI_PLC2_Loi_Dry_Run" )
      S_Coil( "AI_PLC2_Loi_Tong" )
   END_RUNG
   // the same network as SCL:
   IF "AI_PLC2_Loi_Dry_Run" THEN "AI_PLC2_Loi_Tong" := TRUE; END_IF;
END_REGION

REGION Network 79: Tổng hợp lỗi PLC2 từ AI_PLC2_Loi_Dosing
   RUNG wire#powerrail
      Contact( "AI_PLC2_Loi_Dosing" )
      S_Coil( "AI_PLC2_Loi_Tong" )
   END_RUNG
   // the same network as SCL:
   IF "AI_PLC2_Loi_Dosing" THEN "AI_PLC2_Loi_Tong" := TRUE; END_IF;
END_REGION

REGION Network 80: Tổng hợp lỗi PLC2 từ AI_PLC2_Loi_Truyen_Thong
   RUNG wire#powerrail
      Contact( "AI_PLC2_Loi_Truyen_Thong" )
      S_Coil( "AI_PLC2_Loi_Tong" )
   END_RUNG
   // the same network as SCL:
   IF "AI_PLC2_Loi_Truyen_Thong" THEN "AI_PLC2_Loi_Tong" := TRUE; END_IF;
END_REGION

REGION Network 81: Tổng hợp lỗi PLC2 từ AI_PLC2_Loi_Setpoint
   RUNG wire#powerrail
      Contact( "AI_PLC2_Loi_Setpoint" )
      S_Coil( "AI_PLC2_Loi_Tong" )
   END_RUNG
   // the same network as SCL:
   IF "AI_PLC2_Loi_Setpoint" THEN "AI_PLC2_Loi_Tong" := TRUE; END_IF;
END_REGION

REGION Network 82: Reset AI_PLC2_Loi_Tong từ nút vật lý
   RUNG wire#powerrail
      Contact( "AI_Nut_Reset_Nhan_Eff" )
      I_Contact( "AI_PLC2_EStop_Latch" )
      I_Contact( "AI_Nut_EStop_Nhan_Eff" )
      R_Coil( "AI_PLC2_Loi_Tong" )
   END_RUNG
   // the same network as SCL:
   IF "AI_Nut_Reset_Nhan_Eff" AND NOT "AI_PLC2_EStop_Latch" AND NOT "AI_Nut_EStop_Nhan_Eff" THEN
       "AI_PLC2_Loi_Tong" := FALSE;
   END_IF;
END_REGION

REGION Network 83: Reset AI_PLC2_Loi_Dry_Run từ nút vật lý
   RUNG wire#powerrail
      Contact( "AI_Nut_Reset_Nhan_Eff" )
      I_Contact( "AI_PLC2_EStop_Latch" )
      I_Contact( "AI_Nut_EStop_Nhan_Eff" )
      R_Coil( "AI_PLC2_Loi_Dry_Run" )
   END_RUNG
   // the same network as SCL:
   IF "AI_Nut_Reset_Nhan_Eff" AND NOT "AI_PLC2_EStop_Latch" AND NOT "AI_Nut_EStop_Nhan_Eff" THEN
       "AI_PLC2_Loi_Dry_Run" := FALSE;
   END_IF;
END_REGION

REGION Network 84: Reset AI_PLC2_Loi_Dosing từ nút vật lý
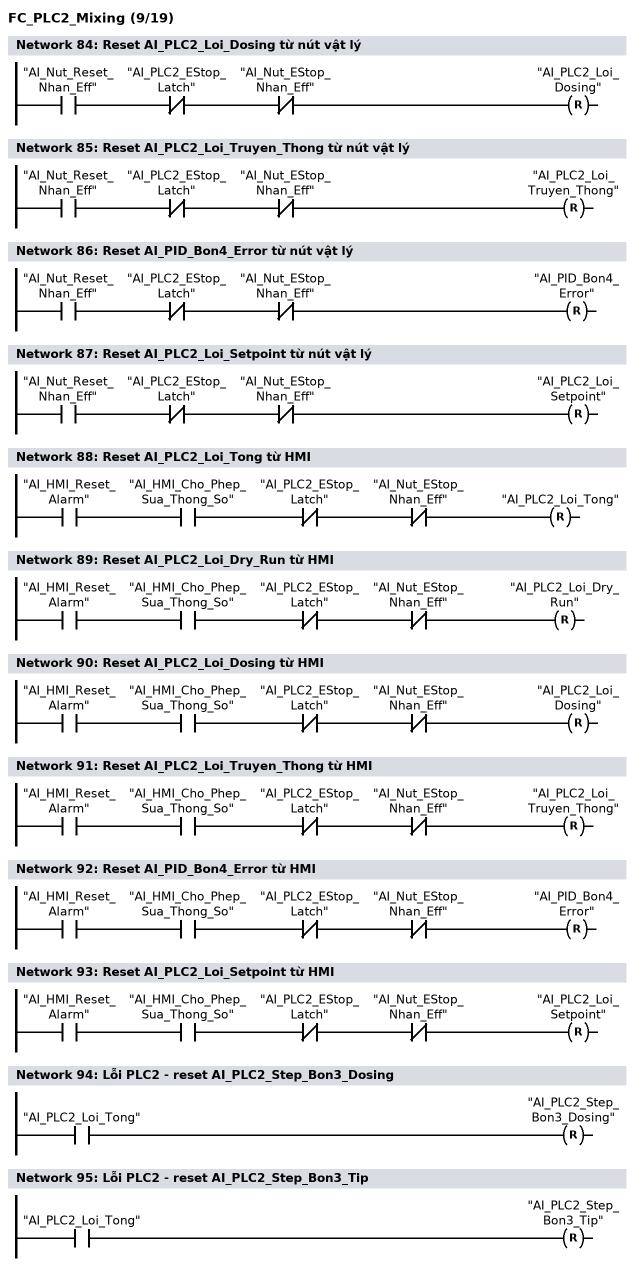
   RUNG wire#powerrail
      Contact( "AI_Nut_Reset_Nhan_Eff" )
      I_Contact( "AI_PLC2_EStop_Latch" )
      I_Contact( "AI_Nut_EStop_Nhan_Eff" )
      R_Coil( "AI_PLC2_Loi_Dosing" )
   END_RUNG
   // the same network as SCL:
   IF "AI_Nut_Reset_Nhan_Eff" AND NOT "AI_PLC2_EStop_Latch" AND NOT "AI_Nut_EStop_Nhan_Eff" THEN
       "AI_PLC2_Loi_Dosing" := FALSE;
   END_IF;
END_REGION

REGION Network 85: Reset AI_PLC2_Loi_Truyen_Thong từ nút vật lý
   RUNG wire#powerrail
      Contact( "AI_Nut_Reset_Nhan_Eff" )
      I_Contact( "AI_PLC2_EStop_Latch" )
      I_Contact( "AI_Nut_EStop_Nhan_Eff" )
      R_Coil( "AI_PLC2_Loi_Truyen_Thong" )
   END_RUNG
   // the same network as SCL:
   IF "AI_Nut_Reset_Nhan_Eff" AND NOT "AI_PLC2_EStop_Latch" AND NOT "AI_Nut_EStop_Nhan_Eff" THEN
       "AI_PLC2_Loi_Truyen_Thong" := FALSE;
   END_IF;
END_REGION

REGION Network 86: Reset AI_PID_Bon4_Error từ nút vật lý
   RUNG wire#powerrail
      Contact( "AI_Nut_Reset_Nhan_Eff" )
      I_Contact( "AI_PLC2_EStop_Latch" )
      I_Contact( "AI_Nut_EStop_Nhan_Eff" )
      R_Coil( "AI_PID_Bon4_Error" )
   END_RUNG
   // the same network as SCL:
   IF "AI_Nut_Reset_Nhan_Eff" AND NOT "AI_PLC2_EStop_Latch" AND NOT "AI_Nut_EStop_Nhan_Eff" THEN
       "AI_PID_Bon4_Error" := FALSE;
   END_IF;
END_REGION

REGION Network 87: Reset AI_PLC2_Loi_Setpoint từ nút vật lý
   RUNG wire#powerrail
      Contact( "AI_Nut_Reset_Nhan_Eff" )
      I_Contact( "AI_PLC2_EStop_Latch" )
      I_Contact( "AI_Nut_EStop_Nhan_Eff" )
      R_Coil( "AI_PLC2_Loi_Setpoint" )
   END_RUNG
   // the same network as SCL:
   IF "AI_Nut_Reset_Nhan_Eff" AND NOT "AI_PLC2_EStop_Latch" AND NOT "AI_Nut_EStop_Nhan_Eff" THEN
       "AI_PLC2_Loi_Setpoint" := FALSE;
   END_IF;
END_REGION

REGION Network 88: Reset AI_PLC2_Loi_Tong từ HMI
   RUNG wire#powerrail
      Contact( "AI_HMI_Reset_Alarm" )
      Contact( "AI_HMI_Cho_Phep_Sua_Thong_So" )
      I_Contact( "AI_PLC2_EStop_Latch" )
      I_Contact( "AI_Nut_EStop_Nhan_Eff" )
      R_Coil( "AI_PLC2_Loi_Tong" )
   END_RUNG
   // the same network as SCL:
   IF "AI_HMI_Reset_Alarm" AND "AI_HMI_Cho_Phep_Sua_Thong_So" AND NOT "AI_PLC2_EStop_Latch" AND NOT "AI_Nut_EStop_Nhan_Eff" THEN
       "AI_PLC2_Loi_Tong" := FALSE;
   END_IF;
END_REGION

REGION Network 89: Reset AI_PLC2_Loi_Dry_Run từ HMI
   RUNG wire#powerrail
      Contact( "AI_HMI_Reset_Alarm" )
      Contact( "AI_HMI_Cho_Phep_Sua_Thong_So" )
      I_Contact( "AI_PLC2_EStop_Latch" )
      I_Contact( "AI_Nut_EStop_Nhan_Eff" )
      R_Coil( "AI_PLC2_Loi_Dry_Run" )
   END_RUNG
   // the same network as SCL:
   IF "AI_HMI_Reset_Alarm" AND "AI_HMI_Cho_Phep_Sua_Thong_So" AND NOT "AI_PLC2_EStop_Latch" AND NOT "AI_Nut_EStop_Nhan_Eff" THEN
       "AI_PLC2_Loi_Dry_Run" := FALSE;
   END_IF;
END_REGION

REGION Network 90: Reset AI_PLC2_Loi_Dosing từ HMI
   RUNG wire#powerrail
      Contact( "AI_HMI_Reset_Alarm" )
      Contact( "AI_HMI_Cho_Phep_Sua_Thong_So" )
      I_Contact( "AI_PLC2_EStop_Latch" )
      I_Contact( "AI_Nut_EStop_Nhan_Eff" )
      R_Coil( "AI_PLC2_Loi_Dosing" )
   END_RUNG
   // the same network as SCL:
   IF "AI_HMI_Reset_Alarm" AND "AI_HMI_Cho_Phep_Sua_Thong_So" AND NOT "AI_PLC2_EStop_Latch" AND NOT "AI_Nut_EStop_Nhan_Eff" THEN
       "AI_PLC2_Loi_Dosing" := FALSE;
   END_IF;
END_REGION

REGION Network 91: Reset AI_PLC2_Loi_Truyen_Thong từ HMI
   RUNG wire#powerrail
      Contact( "AI_HMI_Reset_Alarm" )
      Contact( "AI_HMI_Cho_Phep_Sua_Thong_So" )
      I_Contact( "AI_PLC2_EStop_Latch" )
      I_Contact( "AI_Nut_EStop_Nhan_Eff" )
      R_Coil( "AI_PLC2_Loi_Truyen_Thong" )
   END_RUNG
   // the same network as SCL:
   IF "AI_HMI_Reset_Alarm" AND "AI_HMI_Cho_Phep_Sua_Thong_So" AND NOT "AI_PLC2_EStop_Latch" AND NOT "AI_Nut_EStop_Nhan_Eff" THEN
       "AI_PLC2_Loi_Truyen_Thong" := FALSE;
   END_IF;
END_REGION

REGION Network 92: Reset AI_PID_Bon4_Error từ HMI
   RUNG wire#powerrail
      Contact( "AI_HMI_Reset_Alarm" )
      Contact( "AI_HMI_Cho_Phep_Sua_Thong_So" )
      I_Contact( "AI_PLC2_EStop_Latch" )
      I_Contact( "AI_Nut_EStop_Nhan_Eff" )
      R_Coil( "AI_PID_Bon4_Error" )
   END_RUNG
   // the same network as SCL:
   IF "AI_HMI_Reset_Alarm" AND "AI_HMI_Cho_Phep_Sua_Thong_So" AND NOT "AI_PLC2_EStop_Latch" AND NOT "AI_Nut_EStop_Nhan_Eff" THEN
       "AI_PID_Bon4_Error" := FALSE;
   END_IF;
END_REGION

REGION Network 93: Reset AI_PLC2_Loi_Setpoint từ HMI
   RUNG wire#powerrail
      Contact( "AI_HMI_Reset_Alarm" )
      Contact( "AI_HMI_Cho_Phep_Sua_Thong_So" )
      I_Contact( "AI_PLC2_EStop_Latch" )
      I_Contact( "AI_Nut_EStop_Nhan_Eff" )
      R_Coil( "AI_PLC2_Loi_Setpoint" )
   END_RUNG
   // the same network as SCL:
   IF "AI_HMI_Reset_Alarm" AND "AI_HMI_Cho_Phep_Sua_Thong_So" AND NOT "AI_PLC2_EStop_Latch" AND NOT "AI_Nut_EStop_Nhan_Eff" THEN
       "AI_PLC2_Loi_Setpoint" := FALSE;
   END_IF;
END_REGION

REGION Network 94: Lỗi PLC2 - reset AI_PLC2_Step_Bon3_Dosing
   RUNG wire#powerrail
      Contact( "AI_PLC2_Loi_Tong" )
      R_Coil( "AI_PLC2_Step_Bon3_Dosing" )
   END_RUNG
   // the same network as SCL:
   IF "AI_PLC2_Loi_Tong" THEN "AI_PLC2_Step_Bon3_Dosing" := FALSE; END_IF;
END_REGION

REGION Network 95: Lỗi PLC2 - reset AI_PLC2_Step_Bon3_Tip
   RUNG wire#powerrail
      Contact( "AI_PLC2_Loi_Tong" )
      R_Coil( "AI_PLC2_Step_Bon3_Tip" )
   END_RUNG
   // the same network as SCL:
   IF "AI_PLC2_Loi_Tong" THEN "AI_PLC2_Step_Bon3_Tip" := FALSE; END_IF;
END_REGION

REGION Network 96: Lỗi PLC2 - reset AI_PLC2_Step_Bon3_Khuay
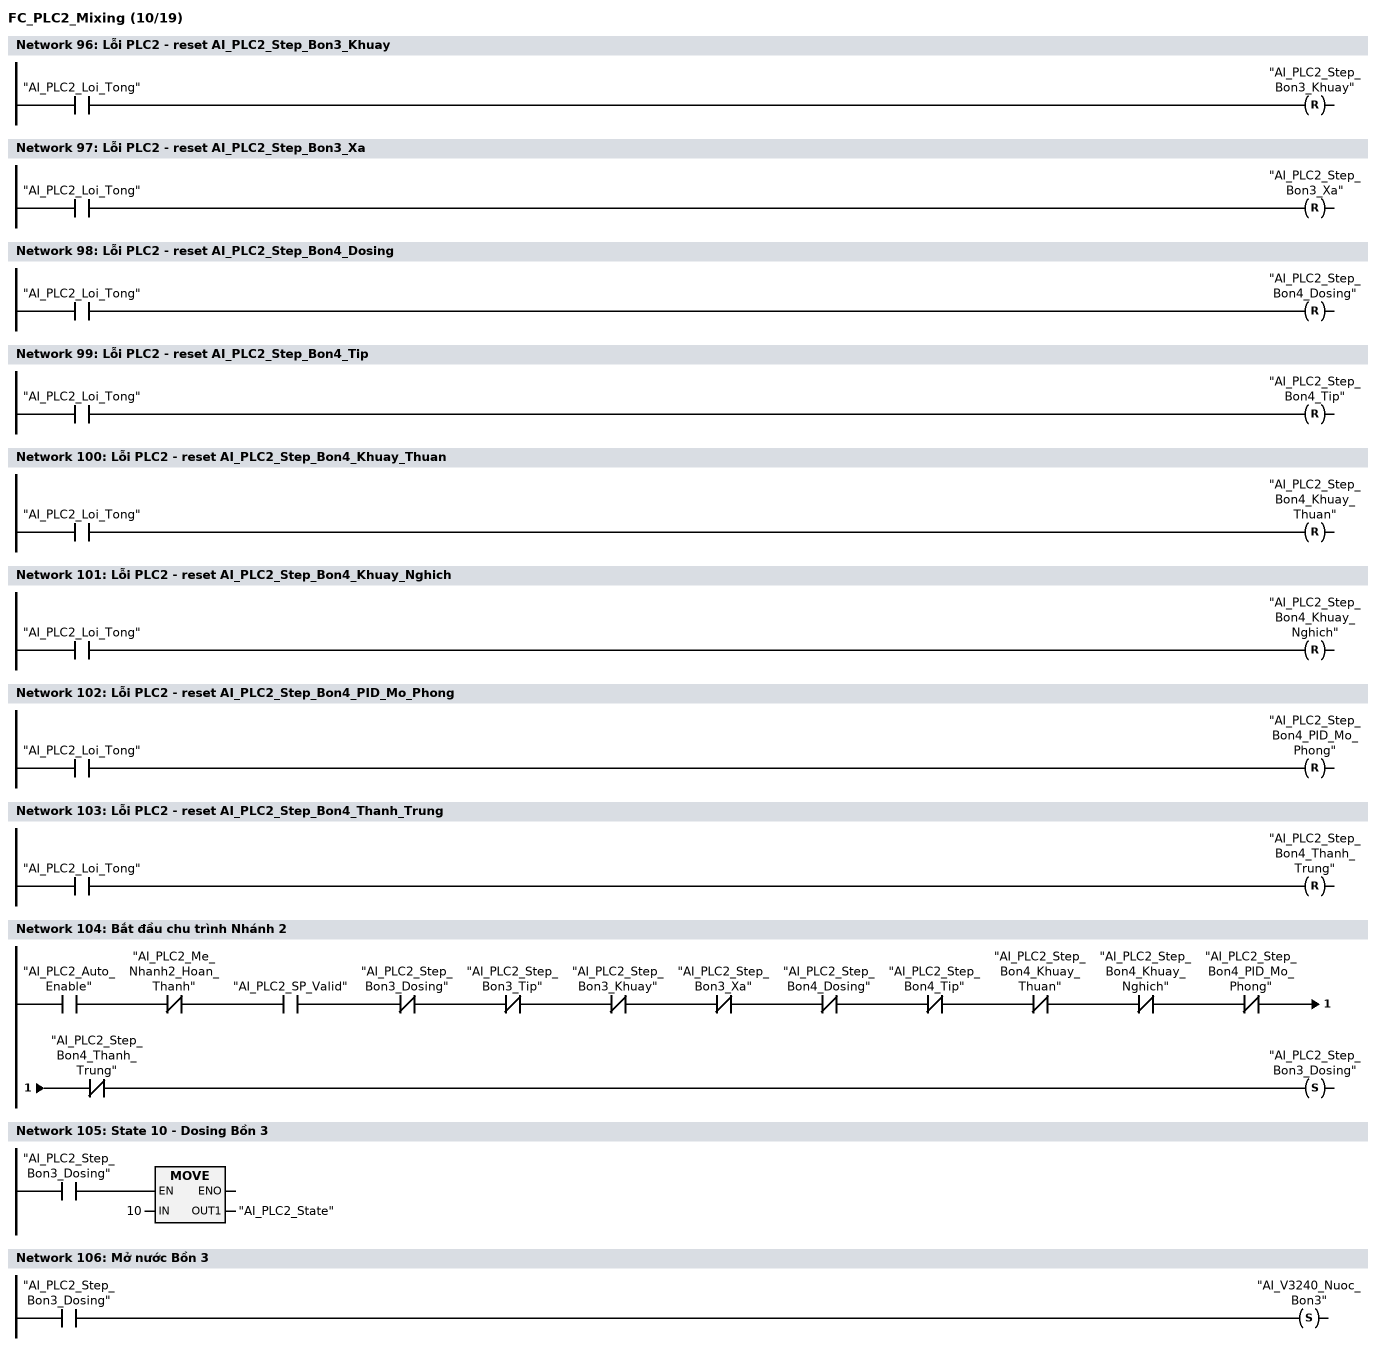
   RUNG wire#powerrail
      Contact( "AI_PLC2_Loi_Tong" )
      R_Coil( "AI_PLC2_Step_Bon3_Khuay" )
   END_RUNG
   // the same network as SCL:
   IF "AI_PLC2_Loi_Tong" THEN "AI_PLC2_Step_Bon3_Khuay" := FALSE; END_IF;
END_REGION

REGION Network 97: Lỗi PLC2 - reset AI_PLC2_Step_Bon3_Xa
   RUNG wire#powerrail
      Contact( "AI_PLC2_Loi_Tong" )
      R_Coil( "AI_PLC2_Step_Bon3_Xa" )
   END_RUNG
   // the same network as SCL:
   IF "AI_PLC2_Loi_Tong" THEN "AI_PLC2_Step_Bon3_Xa" := FALSE; END_IF;
END_REGION

REGION Network 98: Lỗi PLC2 - reset AI_PLC2_Step_Bon4_Dosing
   RUNG wire#powerrail
      Contact( "AI_PLC2_Loi_Tong" )
      R_Coil( "AI_PLC2_Step_Bon4_Dosing" )
   END_RUNG
   // the same network as SCL:
   IF "AI_PLC2_Loi_Tong" THEN "AI_PLC2_Step_Bon4_Dosing" := FALSE; END_IF;
END_REGION

REGION Network 99: Lỗi PLC2 - reset AI_PLC2_Step_Bon4_Tip
   RUNG wire#powerrail
      Contact( "AI_PLC2_Loi_Tong" )
      R_Coil( "AI_PLC2_Step_Bon4_Tip" )
   END_RUNG
   // the same network as SCL:
   IF "AI_PLC2_Loi_Tong" THEN "AI_PLC2_Step_Bon4_Tip" := FALSE; END_IF;
END_REGION

REGION Network 100: Lỗi PLC2 - reset AI_PLC2_Step_Bon4_Khuay_Thuan
   RUNG wire#powerrail
      Contact( "AI_PLC2_Loi_Tong" )
      R_Coil( "AI_PLC2_Step_Bon4_Khuay_Thuan" )
   END_RUNG
   // the same network as SCL:
   IF "AI_PLC2_Loi_Tong" THEN "AI_PLC2_Step_Bon4_Khuay_Thuan" := FALSE; END_IF;
END_REGION

REGION Network 101: Lỗi PLC2 - reset AI_PLC2_Step_Bon4_Khuay_Nghich
   RUNG wire#powerrail
      Contact( "AI_PLC2_Loi_Tong" )
      R_Coil( "AI_PLC2_Step_Bon4_Khuay_Nghich" )
   END_RUNG
   // the same network as SCL:
   IF "AI_PLC2_Loi_Tong" THEN "AI_PLC2_Step_Bon4_Khuay_Nghich" := FALSE; END_IF;
END_REGION

REGION Network 102: Lỗi PLC2 - reset AI_PLC2_Step_Bon4_PID_Mo_Phong
   RUNG wire#powerrail
      Contact( "AI_PLC2_Loi_Tong" )
      R_Coil( "AI_PLC2_Step_Bon4_PID_Mo_Phong" )
   END_RUNG
   // the same network as SCL:
   IF "AI_PLC2_Loi_Tong" THEN "AI_PLC2_Step_Bon4_PID_Mo_Phong" := FALSE; END_IF;
END_REGION

REGION Network 103: Lỗi PLC2 - reset AI_PLC2_Step_Bon4_Thanh_Trung
   RUNG wire#powerrail
      Contact( "AI_PLC2_Loi_Tong" )
      R_Coil( "AI_PLC2_Step_Bon4_Thanh_Trung" )
   END_RUNG
   // the same network as SCL:
   IF "AI_PLC2_Loi_Tong" THEN "AI_PLC2_Step_Bon4_Thanh_Trung" := FALSE; END_IF;
END_REGION

REGION Network 104: Bắt đầu chu trình Nhánh 2
   RUNG wire#powerrail
      Contact( "AI_PLC2_Auto_Enable" )
      I_Contact( "AI_PLC2_Me_Nhanh2_Hoan_Thanh" )
      Contact( "AI_PLC2_SP_Valid" )
      I_Contact( "AI_PLC2_Step_Bon3_Dosing" )
      I_Contact( "AI_PLC2_Step_Bon3_Tip" )
      I_Contact( "AI_PLC2_Step_Bon3_Khuay" )
      I_Contact( "AI_PLC2_Step_Bon3_Xa" )
      I_Contact( "AI_PLC2_Step_Bon4_Dosing" )
      I_Contact( "AI_PLC2_Step_Bon4_Tip" )
      I_Contact( "AI_PLC2_Step_Bon4_Khuay_Thuan" )
      I_Contact( "AI_PLC2_Step_Bon4_Khuay_Nghich" )
      I_Contact( "AI_PLC2_Step_Bon4_PID_Mo_Phong" )
      I_Contact( "AI_PLC2_Step_Bon4_Thanh_Trung" )
      S_Coil( "AI_PLC2_Step_Bon3_Dosing" )
   END_RUNG
   // the same network as SCL:
   IF "AI_PLC2_Auto_Enable" AND NOT "AI_PLC2_Me_Nhanh2_Hoan_Thanh" AND "AI_PLC2_SP_Valid" AND NOT "AI_PLC2_Step_Bon3_Dosing" AND NOT "AI_PLC2_Step_Bon3_Tip" AND NOT "AI_PLC2_Step_Bon3_Khuay" AND NOT "AI_PLC2_Step_Bon3_Xa" AND NOT "AI_PLC2_Step_Bon4_Dosing" AND NOT "AI_PLC2_Step_Bon4_Tip" AND NOT "AI_PLC2_Step_Bon4_Khuay_Thuan" AND NOT "AI_PLC2_Step_Bon4_Khuay_Nghich" AND NOT "AI_PLC2_Step_Bon4_PID_Mo_Phong" AND NOT "AI_PLC2_Step_Bon4_Thanh_Trung" THEN
       "AI_PLC2_Step_Bon3_Dosing" := TRUE;
   END_IF;
END_REGION

REGION Network 105: State 10 - Dosing Bồn 3
   RUNG wire#powerrail
      Contact( "AI_PLC2_Step_Bon3_Dosing" )
      { S7_GenerateENO := "TRUE" } Move(in := 10, out1 => "AI_PLC2_State")
   END_RUNG
   // the same network as SCL:
   IF "AI_PLC2_Step_Bon3_Dosing" THEN "AI_PLC2_State" := 10; END_IF;
END_REGION

REGION Network 106: Mở nước Bồn 3
   RUNG wire#powerrail
      Contact( "AI_PLC2_Step_Bon3_Dosing" )
      S_Coil( "AI_V3240_Nuoc_Bon3" )
   END_RUNG
   // the same network as SCL:
   IF "AI_PLC2_Step_Bon3_Dosing" THEN "AI_V3240_Nuoc_Bon3" := TRUE; END_IF;
END_REGION

REGION Network 107: CV nước Bồn 3 mở 100 phần trăm
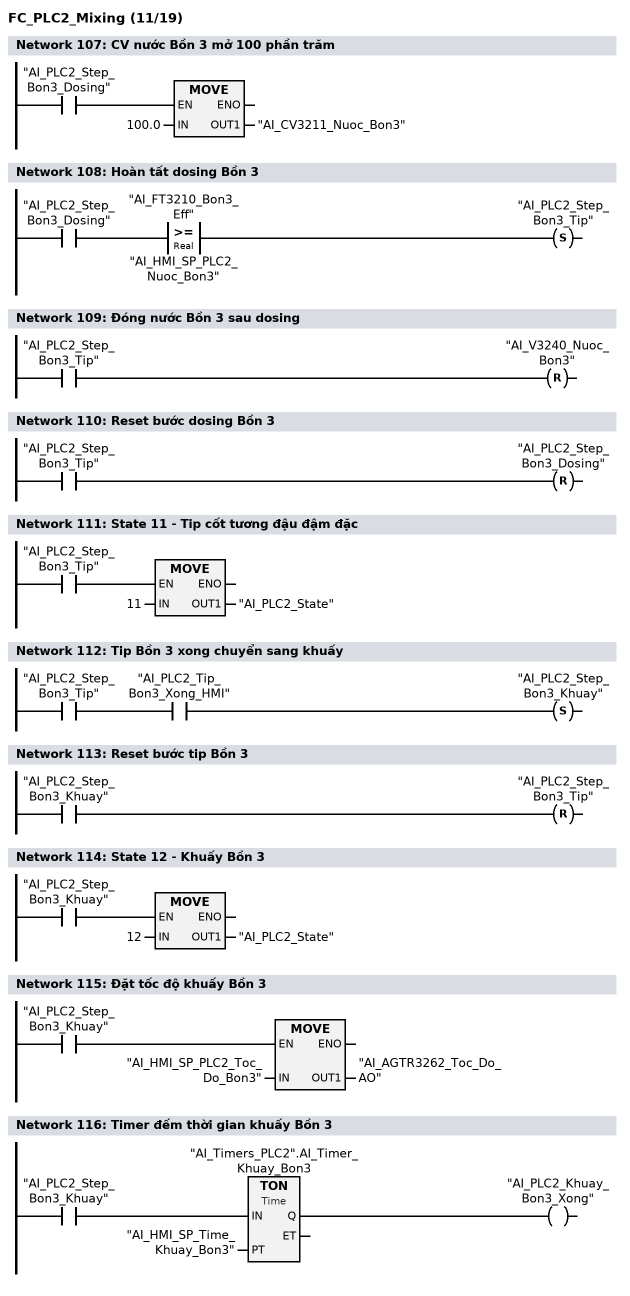
   RUNG wire#powerrail
      Contact( "AI_PLC2_Step_Bon3_Dosing" )
      { S7_GenerateENO := "TRUE" } Move(in := 100.0, out1 => "AI_CV3211_Nuoc_Bon3")
   END_RUNG
   // the same network as SCL:
   IF "AI_PLC2_Step_Bon3_Dosing" THEN "AI_CV3211_Nuoc_Bon3" := 100.0; END_IF;
END_REGION

REGION Network 108: Hoàn tất dosing Bồn 3
   RUNG wire#powerrail
      Contact( "AI_PLC2_Step_Bon3_Dosing" )
      { S7_Templates := "SrcType := Real" } GE_Contact(in1 := "AI_FT3210_Bon3_Eff", in2 := "AI_HMI_SP_PLC2_Nuoc_Bon3")
      S_Coil( "AI_PLC2_Step_Bon3_Tip" )
   END_RUNG
   // the same network as SCL:
   IF "AI_PLC2_Step_Bon3_Dosing" AND ("AI_FT3210_Bon3_Eff" >= "AI_HMI_SP_PLC2_Nuoc_Bon3") THEN
       "AI_PLC2_Step_Bon3_Tip" := TRUE;
   END_IF;
END_REGION

REGION Network 109: Đóng nước Bồn 3 sau dosing
   RUNG wire#powerrail
      Contact( "AI_PLC2_Step_Bon3_Tip" )
      R_Coil( "AI_V3240_Nuoc_Bon3" )
   END_RUNG
   // the same network as SCL:
   IF "AI_PLC2_Step_Bon3_Tip" THEN "AI_V3240_Nuoc_Bon3" := FALSE; END_IF;
END_REGION

REGION Network 110: Reset bước dosing Bồn 3
   RUNG wire#powerrail
      Contact( "AI_PLC2_Step_Bon3_Tip" )
      R_Coil( "AI_PLC2_Step_Bon3_Dosing" )
   END_RUNG
   // the same network as SCL:
   IF "AI_PLC2_Step_Bon3_Tip" THEN "AI_PLC2_Step_Bon3_Dosing" := FALSE; END_IF;
END_REGION

REGION Network 111: State 11 - Tip cốt tương đậu đậm đặc
   RUNG wire#powerrail
      Contact( "AI_PLC2_Step_Bon3_Tip" )
      { S7_GenerateENO := "TRUE" } Move(in := 11, out1 => "AI_PLC2_State")
   END_RUNG
   // the same network as SCL:
   IF "AI_PLC2_Step_Bon3_Tip" THEN "AI_PLC2_State" := 11; END_IF;
END_REGION

REGION Network 112: Tip Bồn 3 xong chuyển sang khuấy
   RUNG wire#powerrail
      Contact( "AI_PLC2_Step_Bon3_Tip" )
      Contact( "AI_PLC2_Tip_Bon3_Xong_HMI" )
      S_Coil( "AI_PLC2_Step_Bon3_Khuay" )
   END_RUNG
   // the same network as SCL:
   IF "AI_PLC2_Step_Bon3_Tip" AND "AI_PLC2_Tip_Bon3_Xong_HMI" THEN "AI_PLC2_Step_Bon3_Khuay" := TRUE; END_IF;
END_REGION

REGION Network 113: Reset bước tip Bồn 3
   RUNG wire#powerrail
      Contact( "AI_PLC2_Step_Bon3_Khuay" )
      R_Coil( "AI_PLC2_Step_Bon3_Tip" )
   END_RUNG
   // the same network as SCL:
   IF "AI_PLC2_Step_Bon3_Khuay" THEN "AI_PLC2_Step_Bon3_Tip" := FALSE; END_IF;
END_REGION

REGION Network 114: State 12 - Khuấy Bồn 3
   RUNG wire#powerrail
      Contact( "AI_PLC2_Step_Bon3_Khuay" )
      { S7_GenerateENO := "TRUE" } Move(in := 12, out1 => "AI_PLC2_State")
   END_RUNG
   // the same network as SCL:
   IF "AI_PLC2_Step_Bon3_Khuay" THEN "AI_PLC2_State" := 12; END_IF;
END_REGION

REGION Network 115: Đặt tốc độ khuấy Bồn 3
   RUNG wire#powerrail
      Contact( "AI_PLC2_Step_Bon3_Khuay" )
      { S7_GenerateENO := "TRUE" } Move(in := "AI_HMI_SP_PLC2_Toc_Do_Bon3", out1 => "AI_AGTR3262_Toc_Do_AO")
   END_RUNG
   // the same network as SCL:
   IF "AI_PLC2_Step_Bon3_Khuay" THEN "AI_AGTR3262_Toc_Do_AO" := "AI_HMI_SP_PLC2_Toc_Do_Bon3"; END_IF;
END_REGION

REGION Network 116: Timer đếm thời gian khuấy Bồn 3
   RUNG wire#powerrail
      Contact( "AI_PLC2_Step_Bon3_Khuay" )
      { S7_Templates := "time_type := Time" } "AI_Timers_PLC2".AI_Timer_Khuay_Bon3.TON(pt := "AI_HMI_SP_Time_Khuay_Bon3", et =>)
      Coil( "AI_PLC2_Khuay_Bon3_Xong" )
   END_RUNG
   // the same network as SCL:
   "AI_Timers_PLC2".AI_Timer_Khuay_Bon3.TON(IN := "AI_PLC2_Step_Bon3_Khuay", PT := "AI_HMI_SP_Time_Khuay_Bon3");
   "AI_PLC2_Khuay_Bon3_Xong" := "AI_Timers_PLC2".AI_Timer_Khuay_Bon3.Q;
END_REGION

REGION Network 117: Khuấy Bồn 3 xong chuyển xả
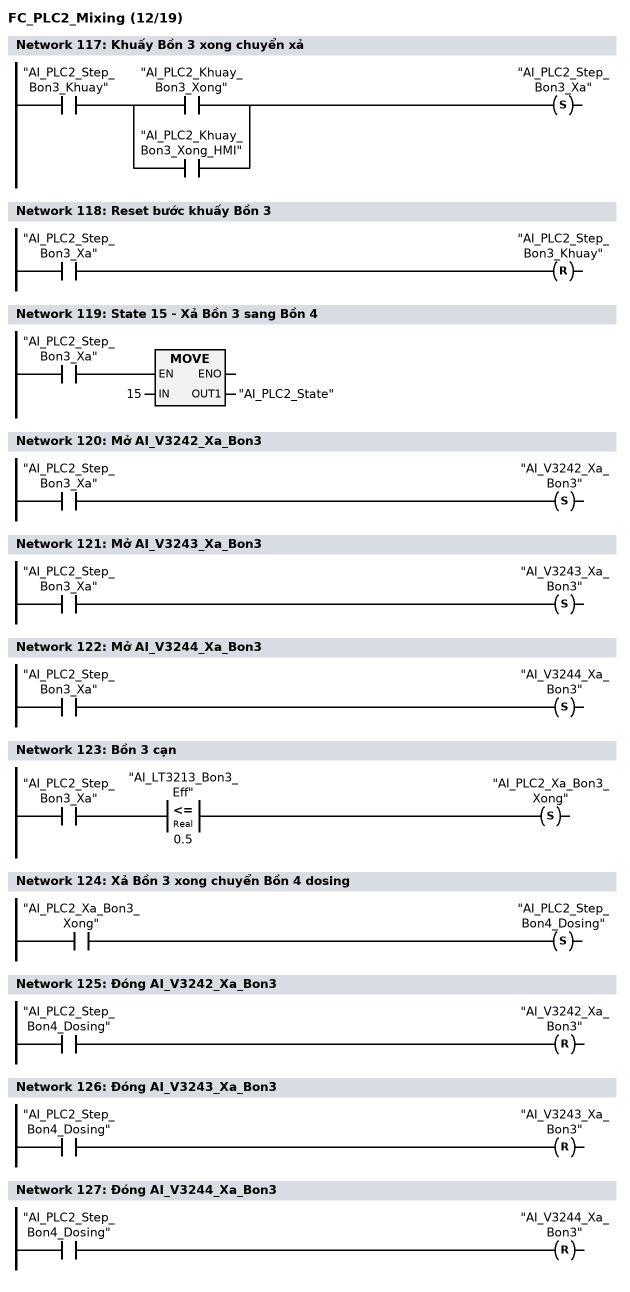
   RUNG wire#powerrail
      Contact( "AI_PLC2_Step_Bon3_Khuay" )
      wire#w1
      Contact( "AI_PLC2_Khuay_Bon3_Xong" )
      wire#w2
      S_Coil( "AI_PLC2_Step_Bon3_Xa" )
   END_RUNG
   RUNG wire#w1
      Contact( "AI_PLC2_Khuay_Bon3_Xong_HMI" )
   END_RUNG wire#w2
   // the same network as SCL:
   IF "AI_PLC2_Step_Bon3_Khuay" AND ("AI_PLC2_Khuay_Bon3_Xong" OR "AI_PLC2_Khuay_Bon3_Xong_HMI") THEN
       "AI_PLC2_Step_Bon3_Xa" := TRUE;
   END_IF;
END_REGION

REGION Network 118: Reset bước khuấy Bồn 3
   RUNG wire#powerrail
      Contact( "AI_PLC2_Step_Bon3_Xa" )
      R_Coil( "AI_PLC2_Step_Bon3_Khuay" )
   END_RUNG
   // the same network as SCL:
   IF "AI_PLC2_Step_Bon3_Xa" THEN "AI_PLC2_Step_Bon3_Khuay" := FALSE; END_IF;
END_REGION

REGION Network 119: State 15 - Xả Bồn 3 sang Bồn 4
   RUNG wire#powerrail
      Contact( "AI_PLC2_Step_Bon3_Xa" )
      { S7_GenerateENO := "TRUE" } Move(in := 15, out1 => "AI_PLC2_State")
   END_RUNG
   // the same network as SCL:
   IF "AI_PLC2_Step_Bon3_Xa" THEN "AI_PLC2_State" := 15; END_IF;
END_REGION

REGION Network 120: Mở AI_V3242_Xa_Bon3
   RUNG wire#powerrail
      Contact( "AI_PLC2_Step_Bon3_Xa" )
      S_Coil( "AI_V3242_Xa_Bon3" )
   END_RUNG
   // the same network as SCL:
   IF "AI_PLC2_Step_Bon3_Xa" THEN "AI_V3242_Xa_Bon3" := TRUE; END_IF;
END_REGION

REGION Network 121: Mở AI_V3243_Xa_Bon3
   RUNG wire#powerrail
      Contact( "AI_PLC2_Step_Bon3_Xa" )
      S_Coil( "AI_V3243_Xa_Bon3" )
   END_RUNG
   // the same network as SCL:
   IF "AI_PLC2_Step_Bon3_Xa" THEN "AI_V3243_Xa_Bon3" := TRUE; END_IF;
END_REGION

REGION Network 122: Mở AI_V3244_Xa_Bon3
   RUNG wire#powerrail
      Contact( "AI_PLC2_Step_Bon3_Xa" )
      S_Coil( "AI_V3244_Xa_Bon3" )
   END_RUNG
   // the same network as SCL:
   IF "AI_PLC2_Step_Bon3_Xa" THEN "AI_V3244_Xa_Bon3" := TRUE; END_IF;
END_REGION

REGION Network 123: Bồn 3 cạn
   RUNG wire#powerrail
      Contact( "AI_PLC2_Step_Bon3_Xa" )
      { S7_Templates := "SrcType := Real" } LE_Contact(in1 := "AI_LT3213_Bon3_Eff", in2 := 0.5)
      S_Coil( "AI_PLC2_Xa_Bon3_Xong" )
   END_RUNG
   // the same network as SCL:
   IF "AI_PLC2_Step_Bon3_Xa" AND ("AI_LT3213_Bon3_Eff" <= 0.5) THEN "AI_PLC2_Xa_Bon3_Xong" := TRUE; END_IF;
END_REGION

REGION Network 124: Xả Bồn 3 xong chuyển Bồn 4 dosing
   RUNG wire#powerrail
      Contact( "AI_PLC2_Xa_Bon3_Xong" )
      S_Coil( "AI_PLC2_Step_Bon4_Dosing" )
   END_RUNG
   // the same network as SCL:
   IF "AI_PLC2_Xa_Bon3_Xong" THEN "AI_PLC2_Step_Bon4_Dosing" := TRUE; END_IF;
END_REGION

REGION Network 125: Đóng AI_V3242_Xa_Bon3
   RUNG wire#powerrail
      Contact( "AI_PLC2_Step_Bon4_Dosing" )
      R_Coil( "AI_V3242_Xa_Bon3" )
   END_RUNG
   // the same network as SCL:
   IF "AI_PLC2_Step_Bon4_Dosing" THEN "AI_V3242_Xa_Bon3" := FALSE; END_IF;
END_REGION

REGION Network 126: Đóng AI_V3243_Xa_Bon3
   RUNG wire#powerrail
      Contact( "AI_PLC2_Step_Bon4_Dosing" )
      R_Coil( "AI_V3243_Xa_Bon3" )
   END_RUNG
   // the same network as SCL:
   IF "AI_PLC2_Step_Bon4_Dosing" THEN "AI_V3243_Xa_Bon3" := FALSE; END_IF;
END_REGION

REGION Network 127: Đóng AI_V3244_Xa_Bon3
   RUNG wire#powerrail
      Contact( "AI_PLC2_Step_Bon4_Dosing" )
      R_Coil( "AI_V3244_Xa_Bon3" )
   END_RUNG
   // the same network as SCL:
   IF "AI_PLC2_Step_Bon4_Dosing" THEN "AI_V3244_Xa_Bon3" := FALSE; END_IF;
END_REGION

REGION Network 128: Reset bước xả Bồn 3
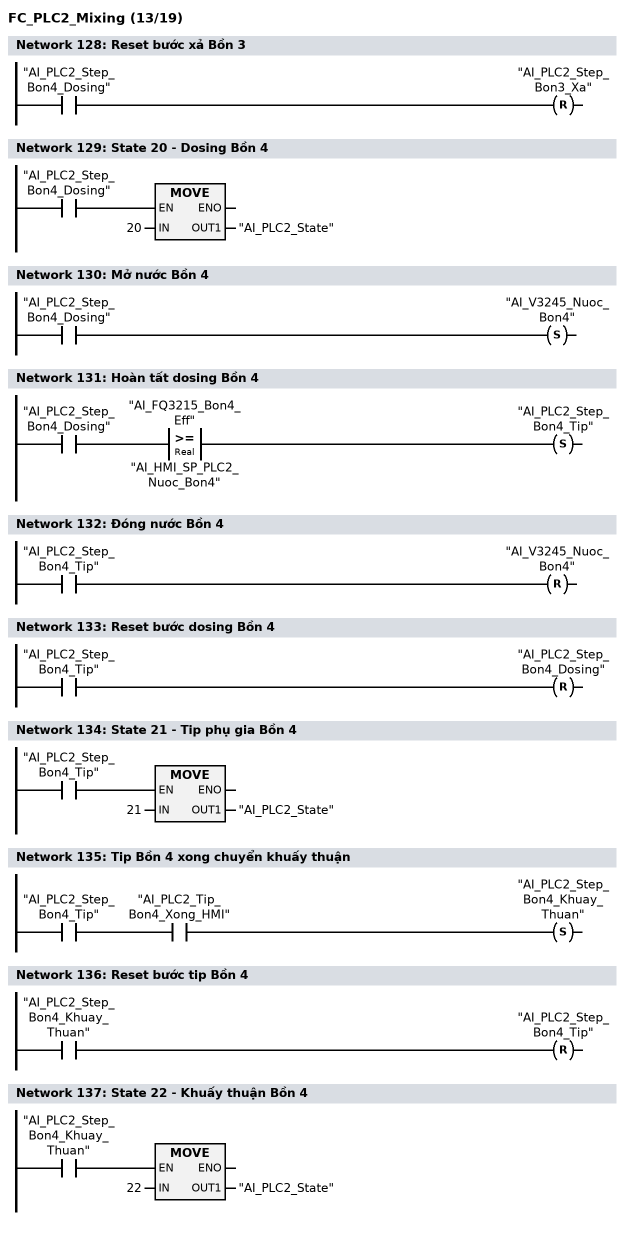
   RUNG wire#powerrail
      Contact( "AI_PLC2_Step_Bon4_Dosing" )
      R_Coil( "AI_PLC2_Step_Bon3_Xa" )
   END_RUNG
   // the same network as SCL:
   IF "AI_PLC2_Step_Bon4_Dosing" THEN "AI_PLC2_Step_Bon3_Xa" := FALSE; END_IF;
END_REGION

REGION Network 129: State 20 - Dosing Bồn 4
   RUNG wire#powerrail
      Contact( "AI_PLC2_Step_Bon4_Dosing" )
      { S7_GenerateENO := "TRUE" } Move(in := 20, out1 => "AI_PLC2_State")
   END_RUNG
   // the same network as SCL:
   IF "AI_PLC2_Step_Bon4_Dosing" THEN "AI_PLC2_State" := 20; END_IF;
END_REGION

REGION Network 130: Mở nước Bồn 4
   RUNG wire#powerrail
      Contact( "AI_PLC2_Step_Bon4_Dosing" )
      S_Coil( "AI_V3245_Nuoc_Bon4" )
   END_RUNG
   // the same network as SCL:
   IF "AI_PLC2_Step_Bon4_Dosing" THEN "AI_V3245_Nuoc_Bon4" := TRUE; END_IF;
END_REGION

REGION Network 131: Hoàn tất dosing Bồn 4
   RUNG wire#powerrail
      Contact( "AI_PLC2_Step_Bon4_Dosing" )
      { S7_Templates := "SrcType := Real" } GE_Contact(in1 := "AI_FQ3215_Bon4_Eff", in2 := "AI_HMI_SP_PLC2_Nuoc_Bon4")
      S_Coil( "AI_PLC2_Step_Bon4_Tip" )
   END_RUNG
   // the same network as SCL:
   IF "AI_PLC2_Step_Bon4_Dosing" AND ("AI_FQ3215_Bon4_Eff" >= "AI_HMI_SP_PLC2_Nuoc_Bon4") THEN
       "AI_PLC2_Step_Bon4_Tip" := TRUE;
   END_IF;
END_REGION

REGION Network 132: Đóng nước Bồn 4
   RUNG wire#powerrail
      Contact( "AI_PLC2_Step_Bon4_Tip" )
      R_Coil( "AI_V3245_Nuoc_Bon4" )
   END_RUNG
   // the same network as SCL:
   IF "AI_PLC2_Step_Bon4_Tip" THEN "AI_V3245_Nuoc_Bon4" := FALSE; END_IF;
END_REGION

REGION Network 133: Reset bước dosing Bồn 4
   RUNG wire#powerrail
      Contact( "AI_PLC2_Step_Bon4_Tip" )
      R_Coil( "AI_PLC2_Step_Bon4_Dosing" )
   END_RUNG
   // the same network as SCL:
   IF "AI_PLC2_Step_Bon4_Tip" THEN "AI_PLC2_Step_Bon4_Dosing" := FALSE; END_IF;
END_REGION

REGION Network 134: State 21 - Tip phụ gia Bồn 4
   RUNG wire#powerrail
      Contact( "AI_PLC2_Step_Bon4_Tip" )
      { S7_GenerateENO := "TRUE" } Move(in := 21, out1 => "AI_PLC2_State")
   END_RUNG
   // the same network as SCL:
   IF "AI_PLC2_Step_Bon4_Tip" THEN "AI_PLC2_State" := 21; END_IF;
END_REGION

REGION Network 135: Tip Bồn 4 xong chuyển khuấy thuận
   RUNG wire#powerrail
      Contact( "AI_PLC2_Step_Bon4_Tip" )
      Contact( "AI_PLC2_Tip_Bon4_Xong_HMI" )
      S_Coil( "AI_PLC2_Step_Bon4_Khuay_Thuan" )
   END_RUNG
   // the same network as SCL:
   IF "AI_PLC2_Step_Bon4_Tip" AND "AI_PLC2_Tip_Bon4_Xong_HMI" THEN
       "AI_PLC2_Step_Bon4_Khuay_Thuan" := TRUE;
   END_IF;
END_REGION

REGION Network 136: Reset bước tip Bồn 4
   RUNG wire#powerrail
      Contact( "AI_PLC2_Step_Bon4_Khuay_Thuan" )
      R_Coil( "AI_PLC2_Step_Bon4_Tip" )
   END_RUNG
   // the same network as SCL:
   IF "AI_PLC2_Step_Bon4_Khuay_Thuan" THEN "AI_PLC2_Step_Bon4_Tip" := FALSE; END_IF;
END_REGION

REGION Network 137: State 22 - Khuấy thuận Bồn 4
   RUNG wire#powerrail
      Contact( "AI_PLC2_Step_Bon4_Khuay_Thuan" )
      { S7_GenerateENO := "TRUE" } Move(in := 22, out1 => "AI_PLC2_State")
   END_RUNG
   // the same network as SCL:
   IF "AI_PLC2_Step_Bon4_Khuay_Thuan" THEN "AI_PLC2_State" := 22; END_IF;
END_REGION

REGION Network 138: Tốc độ khuấy thuận Bồn 4
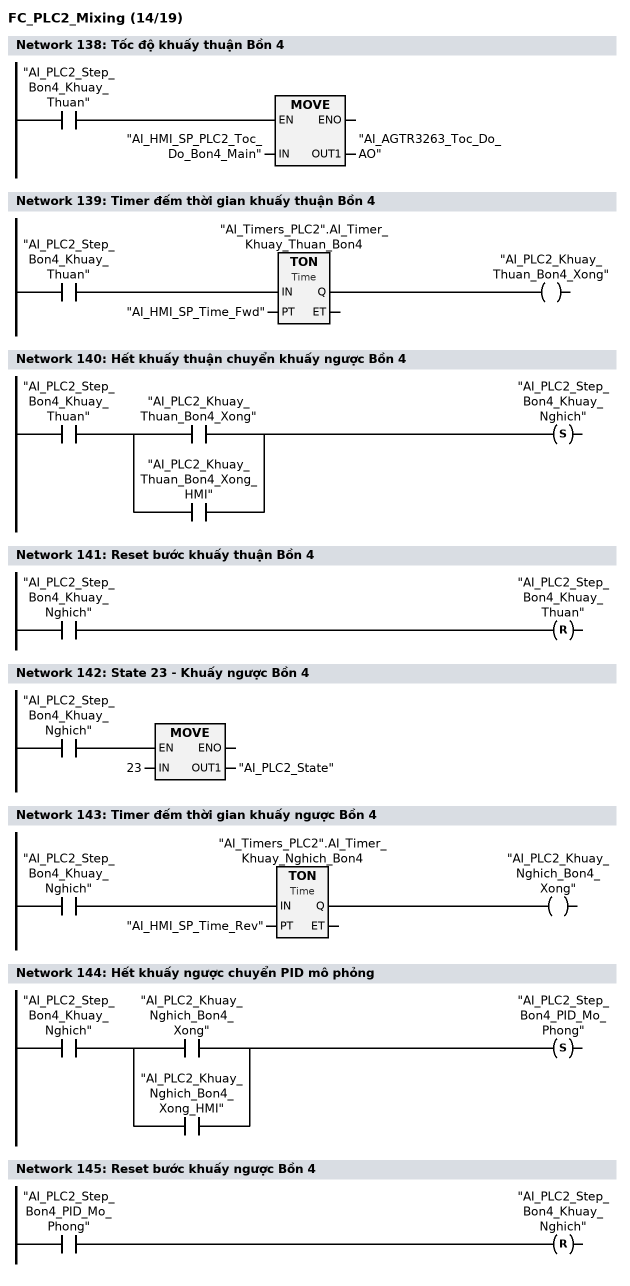
   RUNG wire#powerrail
      Contact( "AI_PLC2_Step_Bon4_Khuay_Thuan" )
      { S7_GenerateENO := "TRUE" } Move(in := "AI_HMI_SP_PLC2_Toc_Do_Bon4_Main", out1 => "AI_AGTR3263_Toc_Do_AO")
   END_RUNG
   // the same network as SCL:
   IF "AI_PLC2_Step_Bon4_Khuay_Thuan" THEN
       "AI_AGTR3263_Toc_Do_AO" := "AI_HMI_SP_PLC2_Toc_Do_Bon4_Main";
   END_IF;
END_REGION

REGION Network 139: Timer đếm thời gian khuấy thuận Bồn 4
   RUNG wire#powerrail
      Contact( "AI_PLC2_Step_Bon4_Khuay_Thuan" )
      { S7_Templates := "time_type := Time" } "AI_Timers_PLC2".AI_Timer_Khuay_Thuan_Bon4.TON(pt := "AI_HMI_SP_Time_Fwd", et =>)
      Coil( "AI_PLC2_Khuay_Thuan_Bon4_Xong" )
   END_RUNG
   // the same network as SCL:
   "AI_Timers_PLC2".AI_Timer_Khuay_Thuan_Bon4.TON(IN := "AI_PLC2_Step_Bon4_Khuay_Thuan",
                           PT := "AI_HMI_SP_Time_Fwd");
   "AI_PLC2_Khuay_Thuan_Bon4_Xong" := "AI_Timers_PLC2".AI_Timer_Khuay_Thuan_Bon4.Q;
END_REGION

REGION Network 140: Hết khuấy thuận chuyển khuấy ngược Bồn 4
   RUNG wire#powerrail
      Contact( "AI_PLC2_Step_Bon4_Khuay_Thuan" )
      wire#w1
      Contact( "AI_PLC2_Khuay_Thuan_Bon4_Xong" )
      wire#w2
      S_Coil( "AI_PLC2_Step_Bon4_Khuay_Nghich" )
   END_RUNG
   RUNG wire#w1
      Contact( "AI_PLC2_Khuay_Thuan_Bon4_Xong_HMI" )
   END_RUNG wire#w2
   // the same network as SCL:
   IF "AI_PLC2_Step_Bon4_Khuay_Thuan" AND ("AI_PLC2_Khuay_Thuan_Bon4_Xong" OR "AI_PLC2_Khuay_Thuan_Bon4_Xong_HMI") THEN
       "AI_PLC2_Step_Bon4_Khuay_Nghich" := TRUE;
   END_IF;
END_REGION

REGION Network 141: Reset bước khuấy thuận Bồn 4
   RUNG wire#powerrail
      Contact( "AI_PLC2_Step_Bon4_Khuay_Nghich" )
      R_Coil( "AI_PLC2_Step_Bon4_Khuay_Thuan" )
   END_RUNG
   // the same network as SCL:
   IF "AI_PLC2_Step_Bon4_Khuay_Nghich" THEN "AI_PLC2_Step_Bon4_Khuay_Thuan" := FALSE; END_IF;
END_REGION

REGION Network 142: State 23 - Khuấy ngược Bồn 4
   RUNG wire#powerrail
      Contact( "AI_PLC2_Step_Bon4_Khuay_Nghich" )
      { S7_GenerateENO := "TRUE" } Move(in := 23, out1 => "AI_PLC2_State")
   END_RUNG
   // the same network as SCL:
   IF "AI_PLC2_Step_Bon4_Khuay_Nghich" THEN "AI_PLC2_State" := 23; END_IF;
END_REGION

REGION Network 143: Timer đếm thời gian khuấy ngược Bồn 4
   RUNG wire#powerrail
      Contact( "AI_PLC2_Step_Bon4_Khuay_Nghich" )
      { S7_Templates := "time_type := Time" } "AI_Timers_PLC2".AI_Timer_Khuay_Nghich_Bon4.TON(pt := "AI_HMI_SP_Time_Rev", et =>)
      Coil( "AI_PLC2_Khuay_Nghich_Bon4_Xong" )
   END_RUNG
   // the same network as SCL:
   "AI_Timers_PLC2".AI_Timer_Khuay_Nghich_Bon4.TON(IN := "AI_PLC2_Step_Bon4_Khuay_Nghich",
                           PT := "AI_HMI_SP_Time_Rev");
   "AI_PLC2_Khuay_Nghich_Bon4_Xong" := "AI_Timers_PLC2".AI_Timer_Khuay_Nghich_Bon4.Q;
END_REGION

REGION Network 144: Hết khuấy ngược chuyển PID mô phỏng
   RUNG wire#powerrail
      Contact( "AI_PLC2_Step_Bon4_Khuay_Nghich" )
      wire#w1
      Contact( "AI_PLC2_Khuay_Nghich_Bon4_Xong" )
      wire#w2
      S_Coil( "AI_PLC2_Step_Bon4_PID_Mo_Phong" )
   END_RUNG
   RUNG wire#w1
      Contact( "AI_PLC2_Khuay_Nghich_Bon4_Xong_HMI" )
   END_RUNG wire#w2
   // the same network as SCL:
   IF "AI_PLC2_Step_Bon4_Khuay_Nghich" AND ("AI_PLC2_Khuay_Nghich_Bon4_Xong" OR "AI_PLC2_Khuay_Nghich_Bon4_Xong_HMI") THEN
       "AI_PLC2_Step_Bon4_PID_Mo_Phong" := TRUE;
   END_IF;
END_REGION

REGION Network 145: Reset bước khuấy ngược Bồn 4
   RUNG wire#powerrail
      Contact( "AI_PLC2_Step_Bon4_PID_Mo_Phong" )
      R_Coil( "AI_PLC2_Step_Bon4_Khuay_Nghich" )
   END_RUNG
   // the same network as SCL:
   IF "AI_PLC2_Step_Bon4_PID_Mo_Phong" THEN "AI_PLC2_Step_Bon4_Khuay_Nghich" := FALSE; END_IF;
END_REGION

REGION Network 146: State 30 - PID mô phỏng Bồn 4
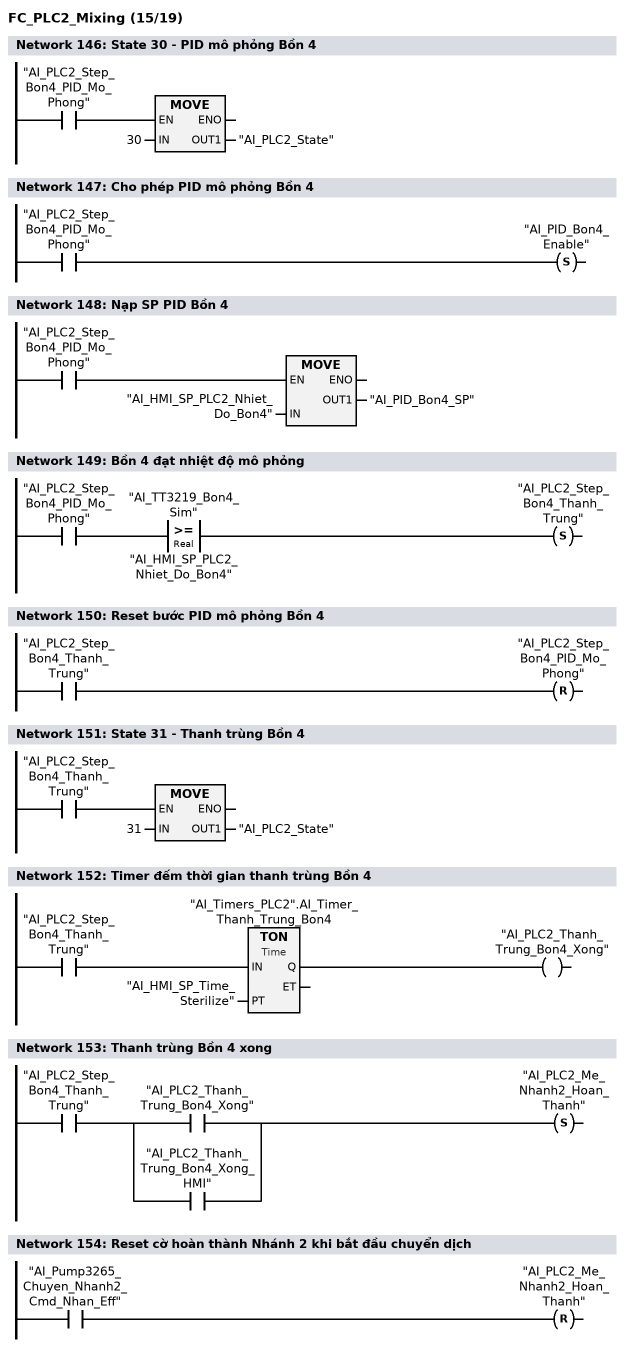
   RUNG wire#powerrail
      Contact( "AI_PLC2_Step_Bon4_PID_Mo_Phong" )
      { S7_GenerateENO := "TRUE" } Move(in := 30, out1 => "AI_PLC2_State")
   END_RUNG
   // the same network as SCL:
   IF "AI_PLC2_Step_Bon4_PID_Mo_Phong" THEN "AI_PLC2_State" := 30; END_IF;
END_REGION

REGION Network 147: Cho phép PID mô phỏng Bồn 4
   RUNG wire#powerrail
      Contact( "AI_PLC2_Step_Bon4_PID_Mo_Phong" )
      S_Coil( "AI_PID_Bon4_Enable" )
   END_RUNG
   // the same network as SCL:
   IF "AI_PLC2_Step_Bon4_PID_Mo_Phong" THEN "AI_PID_Bon4_Enable" := TRUE; END_IF;
END_REGION

REGION Network 148: Nạp SP PID Bồn 4
   RUNG wire#powerrail
      Contact( "AI_PLC2_Step_Bon4_PID_Mo_Phong" )
      { S7_GenerateENO := "TRUE" } Move(in := "AI_HMI_SP_PLC2_Nhiet_Do_Bon4", out1 => "AI_PID_Bon4_SP")
   END_RUNG
   // the same network as SCL:
   IF "AI_PLC2_Step_Bon4_PID_Mo_Phong" THEN "AI_PID_Bon4_SP" := "AI_HMI_SP_PLC2_Nhiet_Do_Bon4"; END_IF;
END_REGION

REGION Network 149: Bồn 4 đạt nhiệt độ mô phỏng
   RUNG wire#powerrail
      Contact( "AI_PLC2_Step_Bon4_PID_Mo_Phong" )
      { S7_Templates := "SrcType := Real" } GE_Contact(in1 := "AI_TT3219_Bon4_Sim", in2 := "AI_HMI_SP_PLC2_Nhiet_Do_Bon4")
      S_Coil( "AI_PLC2_Step_Bon4_Thanh_Trung" )
   END_RUNG
   // the same network as SCL:
   IF "AI_PLC2_Step_Bon4_PID_Mo_Phong" AND ("AI_TT3219_Bon4_Sim" >= "AI_HMI_SP_PLC2_Nhiet_Do_Bon4") THEN
       "AI_PLC2_Step_Bon4_Thanh_Trung" := TRUE;
   END_IF;
END_REGION

REGION Network 150: Reset bước PID mô phỏng Bồn 4
   RUNG wire#powerrail
      Contact( "AI_PLC2_Step_Bon4_Thanh_Trung" )
      R_Coil( "AI_PLC2_Step_Bon4_PID_Mo_Phong" )
   END_RUNG
   // the same network as SCL:
   IF "AI_PLC2_Step_Bon4_Thanh_Trung" THEN "AI_PLC2_Step_Bon4_PID_Mo_Phong" := FALSE; END_IF;
END_REGION

REGION Network 151: State 31 - Thanh trùng Bồn 4
   RUNG wire#powerrail
      Contact( "AI_PLC2_Step_Bon4_Thanh_Trung" )
      { S7_GenerateENO := "TRUE" } Move(in := 31, out1 => "AI_PLC2_State")
   END_RUNG
   // the same network as SCL:
   IF "AI_PLC2_Step_Bon4_Thanh_Trung" THEN "AI_PLC2_State" := 31; END_IF;
END_REGION

REGION Network 152: Timer đếm thời gian thanh trùng Bồn 4
   RUNG wire#powerrail
      Contact( "AI_PLC2_Step_Bon4_Thanh_Trung" )
      { S7_Templates := "time_type := Time" } "AI_Timers_PLC2".AI_Timer_Thanh_Trung_Bon4.TON(pt := "AI_HMI_SP_Time_Sterilize", et =>)
      Coil( "AI_PLC2_Thanh_Trung_Bon4_Xong" )
   END_RUNG
   // the same network as SCL:
   "AI_Timers_PLC2".AI_Timer_Thanh_Trung_Bon4.TON(IN := "AI_PLC2_Step_Bon4_Thanh_Trung",
                           PT := "AI_HMI_SP_Time_Sterilize");
   "AI_PLC2_Thanh_Trung_Bon4_Xong" := "AI_Timers_PLC2".AI_Timer_Thanh_Trung_Bon4.Q;
END_REGION

REGION Network 153: Thanh trùng Bồn 4 xong
   RUNG wire#powerrail
      Contact( "AI_PLC2_Step_Bon4_Thanh_Trung" )
      wire#w1
      Contact( "AI_PLC2_Thanh_Trung_Bon4_Xong" )
      wire#w2
      S_Coil( "AI_PLC2_Me_Nhanh2_Hoan_Thanh" )
   END_RUNG
   RUNG wire#w1
      Contact( "AI_PLC2_Thanh_Trung_Bon4_Xong_HMI" )
   END_RUNG wire#w2
   // the same network as SCL:
   IF "AI_PLC2_Step_Bon4_Thanh_Trung" AND ("AI_PLC2_Thanh_Trung_Bon4_Xong" OR "AI_PLC2_Thanh_Trung_Bon4_Xong_HMI") THEN
       "AI_PLC2_Me_Nhanh2_Hoan_Thanh" := TRUE;
   END_IF;
END_REGION

REGION Network 154: Reset cờ hoàn thành Nhánh 2 khi bắt đầu chuyển dịch
   RUNG wire#powerrail
      Contact( "AI_Pump3265_Chuyen_Nhanh2_Cmd_Nhan_Eff" )
      R_Coil( "AI_PLC2_Me_Nhanh2_Hoan_Thanh" )
   END_RUNG
   // the same network as SCL:
   IF "AI_Pump3265_Chuyen_Nhanh2_Cmd_Nhan_Eff" THEN "AI_PLC2_Me_Nhanh2_Hoan_Thanh" := FALSE; END_IF;
END_REGION

REGION Network 155: Điều khiển bơm chuyển Nhánh 2 từ PLC1
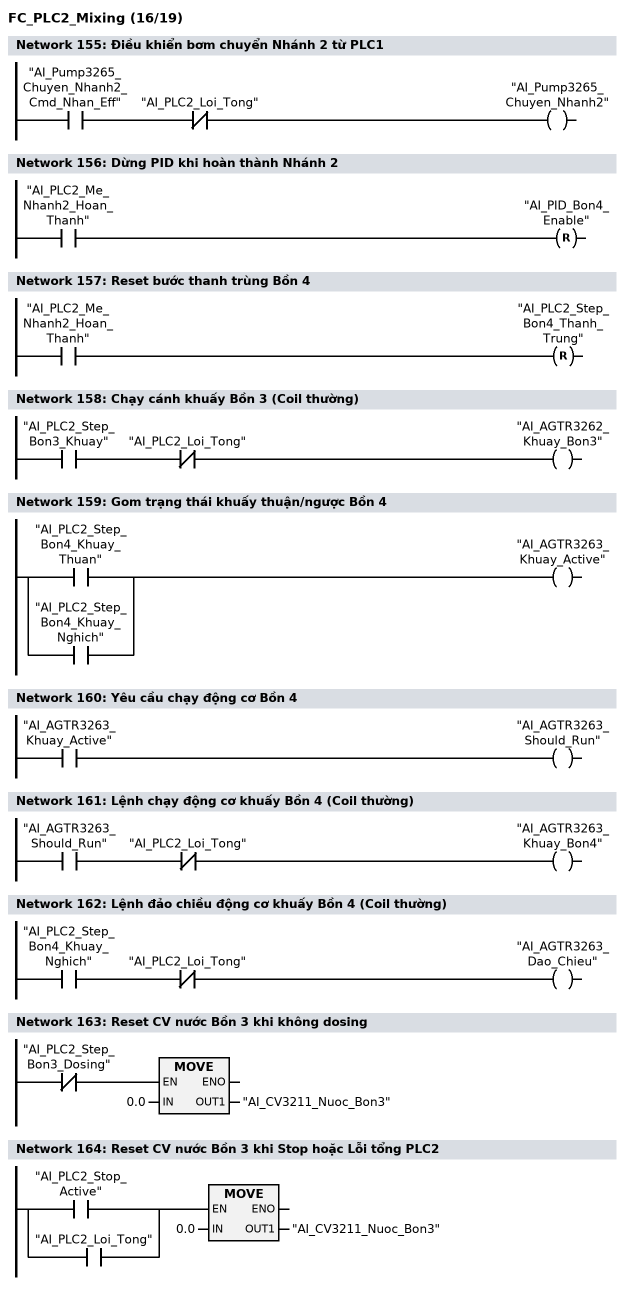
   RUNG wire#powerrail
      Contact( "AI_Pump3265_Chuyen_Nhanh2_Cmd_Nhan_Eff" )
      I_Contact( "AI_PLC2_Loi_Tong" )
      Coil( "AI_Pump3265_Chuyen_Nhanh2" )
   END_RUNG
   // the same network as SCL:
   "AI_Pump3265_Chuyen_Nhanh2" := "AI_Pump3265_Chuyen_Nhanh2_Cmd_Nhan_Eff" AND NOT "AI_PLC2_Loi_Tong";
END_REGION

REGION Network 156: Dừng PID khi hoàn thành Nhánh 2
   RUNG wire#powerrail
      Contact( "AI_PLC2_Me_Nhanh2_Hoan_Thanh" )
      R_Coil( "AI_PID_Bon4_Enable" )
   END_RUNG
   // the same network as SCL:
   IF "AI_PLC2_Me_Nhanh2_Hoan_Thanh" THEN "AI_PID_Bon4_Enable" := FALSE; END_IF;
END_REGION

REGION Network 157: Reset bước thanh trùng Bồn 4
   RUNG wire#powerrail
      Contact( "AI_PLC2_Me_Nhanh2_Hoan_Thanh" )
      R_Coil( "AI_PLC2_Step_Bon4_Thanh_Trung" )
   END_RUNG
   // the same network as SCL:
   IF "AI_PLC2_Me_Nhanh2_Hoan_Thanh" THEN "AI_PLC2_Step_Bon4_Thanh_Trung" := FALSE; END_IF;
END_REGION

REGION Network 158: Chạy cánh khuấy Bồn 3 (Coil thường)
   RUNG wire#powerrail
      Contact( "AI_PLC2_Step_Bon3_Khuay" )
      I_Contact( "AI_PLC2_Loi_Tong" )
      Coil( "AI_AGTR3262_Khuay_Bon3" )
   END_RUNG
   // the same network as SCL:
   "AI_AGTR3262_Khuay_Bon3" := "AI_PLC2_Step_Bon3_Khuay" AND NOT "AI_PLC2_Loi_Tong";
END_REGION

REGION Network 159: Gom trạng thái khuấy thuận/ngược Bồn 4
   RUNG wire#powerrail
      Contact( "AI_PLC2_Step_Bon4_Khuay_Thuan" )
      wire#w1
      Coil( "AI_AGTR3263_Khuay_Active" )
   END_RUNG
   RUNG wire#powerrail
      Contact( "AI_PLC2_Step_Bon4_Khuay_Nghich" )
   END_RUNG wire#w1
   // the same network as SCL:
   "AI_AGTR3263_Khuay_Active" := "AI_PLC2_Step_Bon4_Khuay_Thuan" OR "AI_PLC2_Step_Bon4_Khuay_Nghich";
END_REGION

REGION Network 160: Yêu cầu chạy động cơ Bồn 4
   RUNG wire#powerrail
      Contact( "AI_AGTR3263_Khuay_Active" )
      Coil( "AI_AGTR3263_Should_Run" )
   END_RUNG
   // the same network as SCL:
   "AI_AGTR3263_Should_Run" := "AI_AGTR3263_Khuay_Active";
END_REGION

REGION Network 161: Lệnh chạy động cơ khuấy Bồn 4 (Coil thường)
   RUNG wire#powerrail
      Contact( "AI_AGTR3263_Should_Run" )
      I_Contact( "AI_PLC2_Loi_Tong" )
      Coil( "AI_AGTR3263_Khuay_Bon4" )
   END_RUNG
   // the same network as SCL:
   "AI_AGTR3263_Khuay_Bon4" := "AI_AGTR3263_Should_Run" AND NOT "AI_PLC2_Loi_Tong";
END_REGION

REGION Network 162: Lệnh đảo chiều động cơ khuấy Bồn 4 (Coil thường)
   RUNG wire#powerrail
      Contact( "AI_PLC2_Step_Bon4_Khuay_Nghich" )
      I_Contact( "AI_PLC2_Loi_Tong" )
      Coil( "AI_AGTR3263_Dao_Chieu" )
   END_RUNG
   // the same network as SCL:
   "AI_AGTR3263_Dao_Chieu" := "AI_PLC2_Step_Bon4_Khuay_Nghich" AND NOT "AI_PLC2_Loi_Tong";
END_REGION

REGION Network 163: Reset CV nước Bồn 3 khi không dosing
   RUNG wire#powerrail
      I_Contact( "AI_PLC2_Step_Bon3_Dosing" )
      { S7_GenerateENO := "TRUE" } Move(in := 0.0, out1 => "AI_CV3211_Nuoc_Bon3")
   END_RUNG
   // the same network as SCL:
   IF NOT "AI_PLC2_Step_Bon3_Dosing" THEN "AI_CV3211_Nuoc_Bon3" := 0.0; END_IF;
END_REGION

REGION Network 164: Reset CV nước Bồn 3 khi Stop hoặc Lỗi tổng PLC2
   RUNG wire#powerrail
      Contact( "AI_PLC2_Stop_Active" )
      wire#w1
      { S7_GenerateENO := "TRUE" } Move(in := 0.0, out1 => "AI_CV3211_Nuoc_Bon3")
   END_RUNG
   RUNG wire#powerrail
      Contact( "AI_PLC2_Loi_Tong" )
   END_RUNG wire#w1
   // the same network as SCL:
   IF "AI_PLC2_Stop_Active" OR "AI_PLC2_Loi_Tong" THEN "AI_CV3211_Nuoc_Bon3" := 0.0; END_IF;
END_REGION

REGION Network 165: Clamp CV nước Bồn 3 trong dải 0.0-100.0 (Dưới)
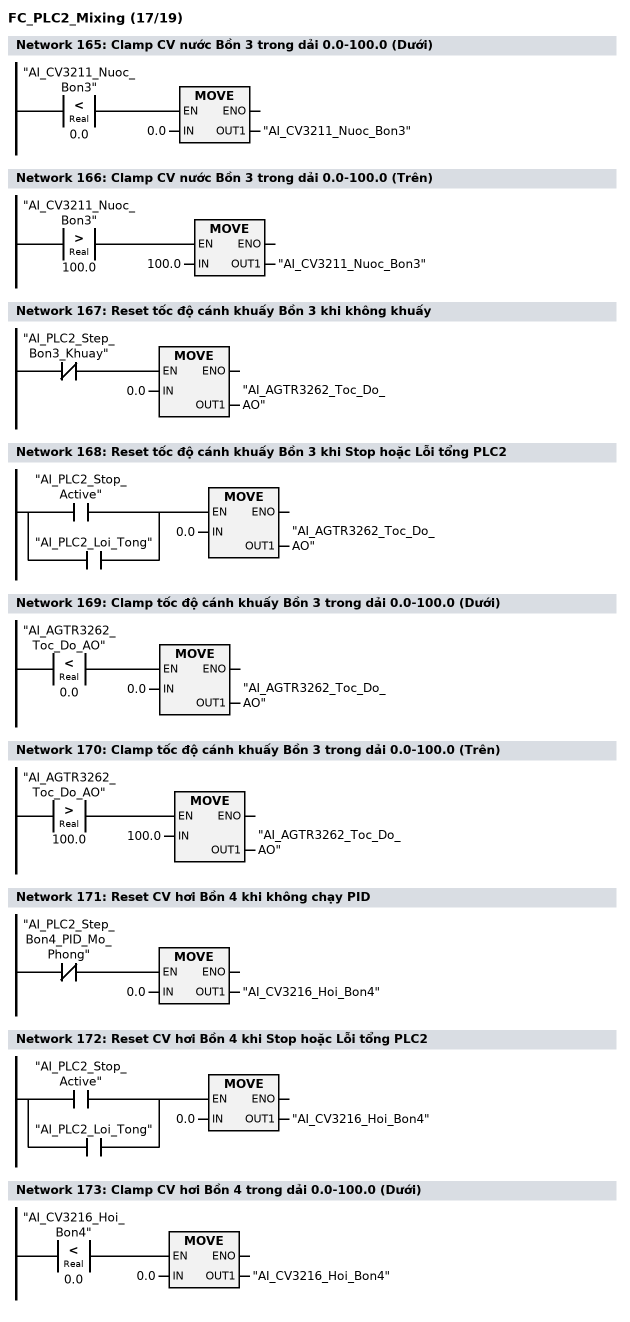
   RUNG wire#powerrail
      { S7_Templates := "SrcType := Real" } LT_Contact(in1 := "AI_CV3211_Nuoc_Bon3", in2 := 0.0)
      { S7_GenerateENO := "TRUE" } Move(in := 0.0, out1 => "AI_CV3211_Nuoc_Bon3")
   END_RUNG
   // the same network as SCL:
   IF "AI_CV3211_Nuoc_Bon3" < 0.0 THEN "AI_CV3211_Nuoc_Bon3" := 0.0; END_IF;
END_REGION

REGION Network 166: Clamp CV nước Bồn 3 trong dải 0.0-100.0 (Trên)
   RUNG wire#powerrail
      { S7_Templates := "SrcType := Real" } GT_Contact(in1 := "AI_CV3211_Nuoc_Bon3", in2 := 100.0)
      { S7_GenerateENO := "TRUE" } Move(in := 100.0, out1 => "AI_CV3211_Nuoc_Bon3")
   END_RUNG
   // the same network as SCL:
   IF "AI_CV3211_Nuoc_Bon3" > 100.0 THEN "AI_CV3211_Nuoc_Bon3" := 100.0; END_IF;
END_REGION

REGION Network 167: Reset tốc độ cánh khuấy Bồn 3 khi không khuấy
   RUNG wire#powerrail
      I_Contact( "AI_PLC2_Step_Bon3_Khuay" )
      { S7_GenerateENO := "TRUE" } Move(in := 0.0, out1 => "AI_AGTR3262_Toc_Do_AO")
   END_RUNG
   // the same network as SCL:
   IF NOT "AI_PLC2_Step_Bon3_Khuay" THEN "AI_AGTR3262_Toc_Do_AO" := 0.0; END_IF;
END_REGION

REGION Network 168: Reset tốc độ cánh khuấy Bồn 3 khi Stop hoặc Lỗi tổng PLC2
   RUNG wire#powerrail
      Contact( "AI_PLC2_Stop_Active" )
      wire#w1
      { S7_GenerateENO := "TRUE" } Move(in := 0.0, out1 => "AI_AGTR3262_Toc_Do_AO")
   END_RUNG
   RUNG wire#powerrail
      Contact( "AI_PLC2_Loi_Tong" )
   END_RUNG wire#w1
   // the same network as SCL:
   IF "AI_PLC2_Stop_Active" OR "AI_PLC2_Loi_Tong" THEN "AI_AGTR3262_Toc_Do_AO" := 0.0; END_IF;
END_REGION

REGION Network 169: Clamp tốc độ cánh khuấy Bồn 3 trong dải 0.0-100.0 (Dưới)
   RUNG wire#powerrail
      { S7_Templates := "SrcType := Real" } LT_Contact(in1 := "AI_AGTR3262_Toc_Do_AO", in2 := 0.0)
      { S7_GenerateENO := "TRUE" } Move(in := 0.0, out1 => "AI_AGTR3262_Toc_Do_AO")
   END_RUNG
   // the same network as SCL:
   IF "AI_AGTR3262_Toc_Do_AO" < 0.0 THEN "AI_AGTR3262_Toc_Do_AO" := 0.0; END_IF;
END_REGION

REGION Network 170: Clamp tốc độ cánh khuấy Bồn 3 trong dải 0.0-100.0 (Trên)
   RUNG wire#powerrail
      { S7_Templates := "SrcType := Real" } GT_Contact(in1 := "AI_AGTR3262_Toc_Do_AO", in2 := 100.0)
      { S7_GenerateENO := "TRUE" } Move(in := 100.0, out1 => "AI_AGTR3262_Toc_Do_AO")
   END_RUNG
   // the same network as SCL:
   IF "AI_AGTR3262_Toc_Do_AO" > 100.0 THEN "AI_AGTR3262_Toc_Do_AO" := 100.0; END_IF;
END_REGION

REGION Network 171: Reset CV hơi Bồn 4 khi không chạy PID
   RUNG wire#powerrail
      I_Contact( "AI_PLC2_Step_Bon4_PID_Mo_Phong" )
      { S7_GenerateENO := "TRUE" } Move(in := 0.0, out1 => "AI_CV3216_Hoi_Bon4")
   END_RUNG
   // the same network as SCL:
   IF NOT "AI_PLC2_Step_Bon4_PID_Mo_Phong" THEN "AI_CV3216_Hoi_Bon4" := 0.0; END_IF;
END_REGION

REGION Network 172: Reset CV hơi Bồn 4 khi Stop hoặc Lỗi tổng PLC2
   RUNG wire#powerrail
      Contact( "AI_PLC2_Stop_Active" )
      wire#w1
      { S7_GenerateENO := "TRUE" } Move(in := 0.0, out1 => "AI_CV3216_Hoi_Bon4")
   END_RUNG
   RUNG wire#powerrail
      Contact( "AI_PLC2_Loi_Tong" )
   END_RUNG wire#w1
   // the same network as SCL:
   IF "AI_PLC2_Stop_Active" OR "AI_PLC2_Loi_Tong" THEN "AI_CV3216_Hoi_Bon4" := 0.0; END_IF;
END_REGION

REGION Network 173: Clamp CV hơi Bồn 4 trong dải 0.0-100.0 (Dưới)
   RUNG wire#powerrail
      { S7_Templates := "SrcType := Real" } LT_Contact(in1 := "AI_CV3216_Hoi_Bon4", in2 := 0.0)
      { S7_GenerateENO := "TRUE" } Move(in := 0.0, out1 => "AI_CV3216_Hoi_Bon4")
   END_RUNG
   // the same network as SCL:
   IF "AI_CV3216_Hoi_Bon4" < 0.0 THEN "AI_CV3216_Hoi_Bon4" := 0.0; END_IF;
END_REGION

REGION Network 174: Clamp CV hơi Bồn 4 trong dải 0.0-100.0 (Trên)
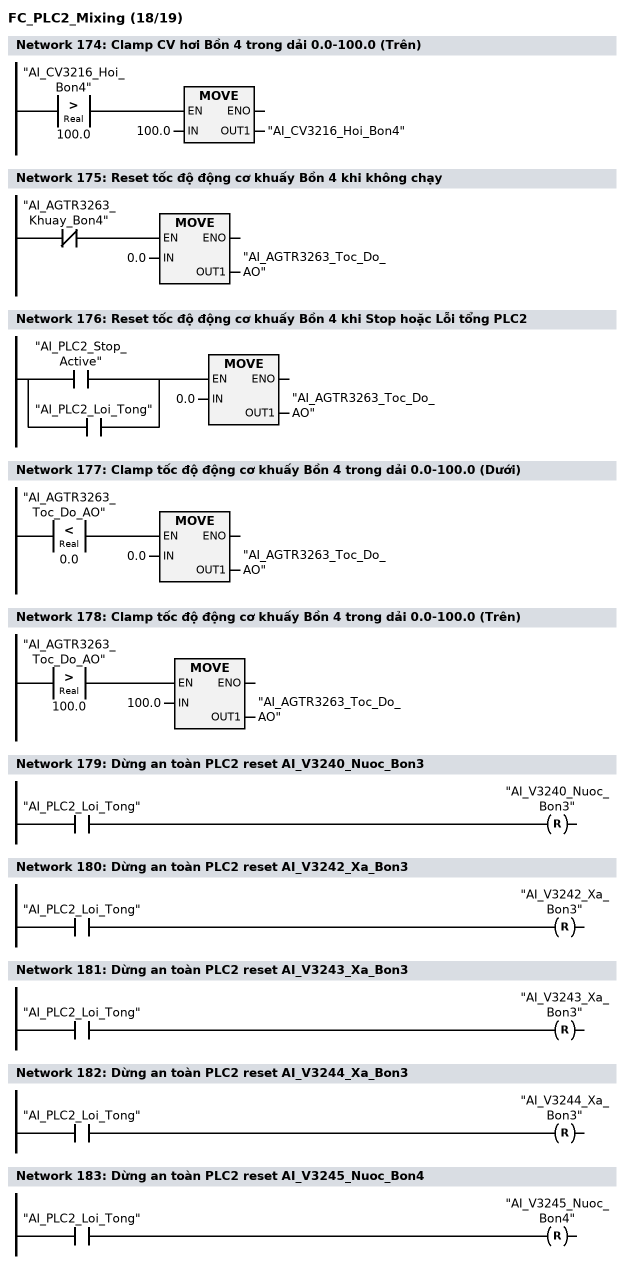
   RUNG wire#powerrail
      { S7_Templates := "SrcType := Real" } GT_Contact(in1 := "AI_CV3216_Hoi_Bon4", in2 := 100.0)
      { S7_GenerateENO := "TRUE" } Move(in := 100.0, out1 => "AI_CV3216_Hoi_Bon4")
   END_RUNG
   // the same network as SCL:
   IF "AI_CV3216_Hoi_Bon4" > 100.0 THEN "AI_CV3216_Hoi_Bon4" := 100.0; END_IF;
END_REGION

REGION Network 175: Reset tốc độ động cơ khuấy Bồn 4 khi không chạy
   RUNG wire#powerrail
      I_Contact( "AI_AGTR3263_Khuay_Bon4" )
      { S7_GenerateENO := "TRUE" } Move(in := 0.0, out1 => "AI_AGTR3263_Toc_Do_AO")
   END_RUNG
   // the same network as SCL:
   IF NOT "AI_AGTR3263_Khuay_Bon4" THEN "AI_AGTR3263_Toc_Do_AO" := 0.0; END_IF;
END_REGION

REGION Network 176: Reset tốc độ động cơ khuấy Bồn 4 khi Stop hoặc Lỗi tổng PLC2
   RUNG wire#powerrail
      Contact( "AI_PLC2_Stop_Active" )
      wire#w1
      { S7_GenerateENO := "TRUE" } Move(in := 0.0, out1 => "AI_AGTR3263_Toc_Do_AO")
   END_RUNG
   RUNG wire#powerrail
      Contact( "AI_PLC2_Loi_Tong" )
   END_RUNG wire#w1
   // the same network as SCL:
   IF "AI_PLC2_Stop_Active" OR "AI_PLC2_Loi_Tong" THEN "AI_AGTR3263_Toc_Do_AO" := 0.0; END_IF;
END_REGION

REGION Network 177: Clamp tốc độ động cơ khuấy Bồn 4 trong dải 0.0-100.0 (Dưới)
   RUNG wire#powerrail
      { S7_Templates := "SrcType := Real" } LT_Contact(in1 := "AI_AGTR3263_Toc_Do_AO", in2 := 0.0)
      { S7_GenerateENO := "TRUE" } Move(in := 0.0, out1 => "AI_AGTR3263_Toc_Do_AO")
   END_RUNG
   // the same network as SCL:
   IF "AI_AGTR3263_Toc_Do_AO" < 0.0 THEN "AI_AGTR3263_Toc_Do_AO" := 0.0; END_IF;
END_REGION

REGION Network 178: Clamp tốc độ động cơ khuấy Bồn 4 trong dải 0.0-100.0 (Trên)
   RUNG wire#powerrail
      { S7_Templates := "SrcType := Real" } GT_Contact(in1 := "AI_AGTR3263_Toc_Do_AO", in2 := 100.0)
      { S7_GenerateENO := "TRUE" } Move(in := 100.0, out1 => "AI_AGTR3263_Toc_Do_AO")
   END_RUNG
   // the same network as SCL:
   IF "AI_AGTR3263_Toc_Do_AO" > 100.0 THEN "AI_AGTR3263_Toc_Do_AO" := 100.0; END_IF;
END_REGION

REGION Network 179: Dừng an toàn PLC2 reset AI_V3240_Nuoc_Bon3
   RUNG wire#powerrail
      Contact( "AI_PLC2_Loi_Tong" )
      R_Coil( "AI_V3240_Nuoc_Bon3" )
   END_RUNG
   // the same network as SCL:
   IF "AI_PLC2_Loi_Tong" THEN "AI_V3240_Nuoc_Bon3" := FALSE; END_IF;
END_REGION

REGION Network 180: Dừng an toàn PLC2 reset AI_V3242_Xa_Bon3
   RUNG wire#powerrail
      Contact( "AI_PLC2_Loi_Tong" )
      R_Coil( "AI_V3242_Xa_Bon3" )
   END_RUNG
   // the same network as SCL:
   IF "AI_PLC2_Loi_Tong" THEN "AI_V3242_Xa_Bon3" := FALSE; END_IF;
END_REGION

REGION Network 181: Dừng an toàn PLC2 reset AI_V3243_Xa_Bon3
   RUNG wire#powerrail
      Contact( "AI_PLC2_Loi_Tong" )
      R_Coil( "AI_V3243_Xa_Bon3" )
   END_RUNG
   // the same network as SCL:
   IF "AI_PLC2_Loi_Tong" THEN "AI_V3243_Xa_Bon3" := FALSE; END_IF;
END_REGION

REGION Network 182: Dừng an toàn PLC2 reset AI_V3244_Xa_Bon3
   RUNG wire#powerrail
      Contact( "AI_PLC2_Loi_Tong" )
      R_Coil( "AI_V3244_Xa_Bon3" )
   END_RUNG
   // the same network as SCL:
   IF "AI_PLC2_Loi_Tong" THEN "AI_V3244_Xa_Bon3" := FALSE; END_IF;
END_REGION

REGION Network 183: Dừng an toàn PLC2 reset AI_V3245_Nuoc_Bon4
   RUNG wire#powerrail
      Contact( "AI_PLC2_Loi_Tong" )
      R_Coil( "AI_V3245_Nuoc_Bon4" )
   END_RUNG
   // the same network as SCL:
   IF "AI_PLC2_Loi_Tong" THEN "AI_V3245_Nuoc_Bon4" := FALSE; END_IF;
END_REGION

REGION Network 184: Dừng an toàn PLC2 reset AI_V3247_Xa_Bon4
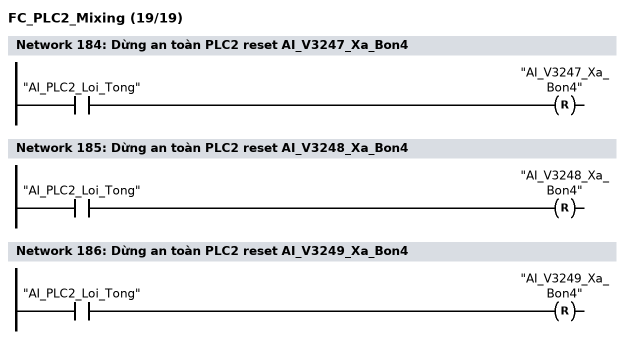
   RUNG wire#powerrail
      Contact( "AI_PLC2_Loi_Tong" )
      R_Coil( "AI_V3247_Xa_Bon4" )
   END_RUNG
   // the same network as SCL:
   IF "AI_PLC2_Loi_Tong" THEN "AI_V3247_Xa_Bon4" := FALSE; END_IF;
END_REGION

REGION Network 185: Dừng an toàn PLC2 reset AI_V3248_Xa_Bon4
   RUNG wire#powerrail
      Contact( "AI_PLC2_Loi_Tong" )
      R_Coil( "AI_V3248_Xa_Bon4" )
   END_RUNG
   // the same network as SCL:
   IF "AI_PLC2_Loi_Tong" THEN "AI_V3248_Xa_Bon4" := FALSE; END_IF;
END_REGION

REGION Network 186: Dừng an toàn PLC2 reset AI_V3249_Xa_Bon4
   RUNG wire#powerrail
      Contact( "AI_PLC2_Loi_Tong" )
      R_Coil( "AI_V3249_Xa_Bon4" )
   END_RUNG
   // the same network as SCL:
   IF "AI_PLC2_Loi_Tong" THEN "AI_V3249_Xa_Bon4" := FALSE; END_IF;
END_REGION
END_FUNCTION
